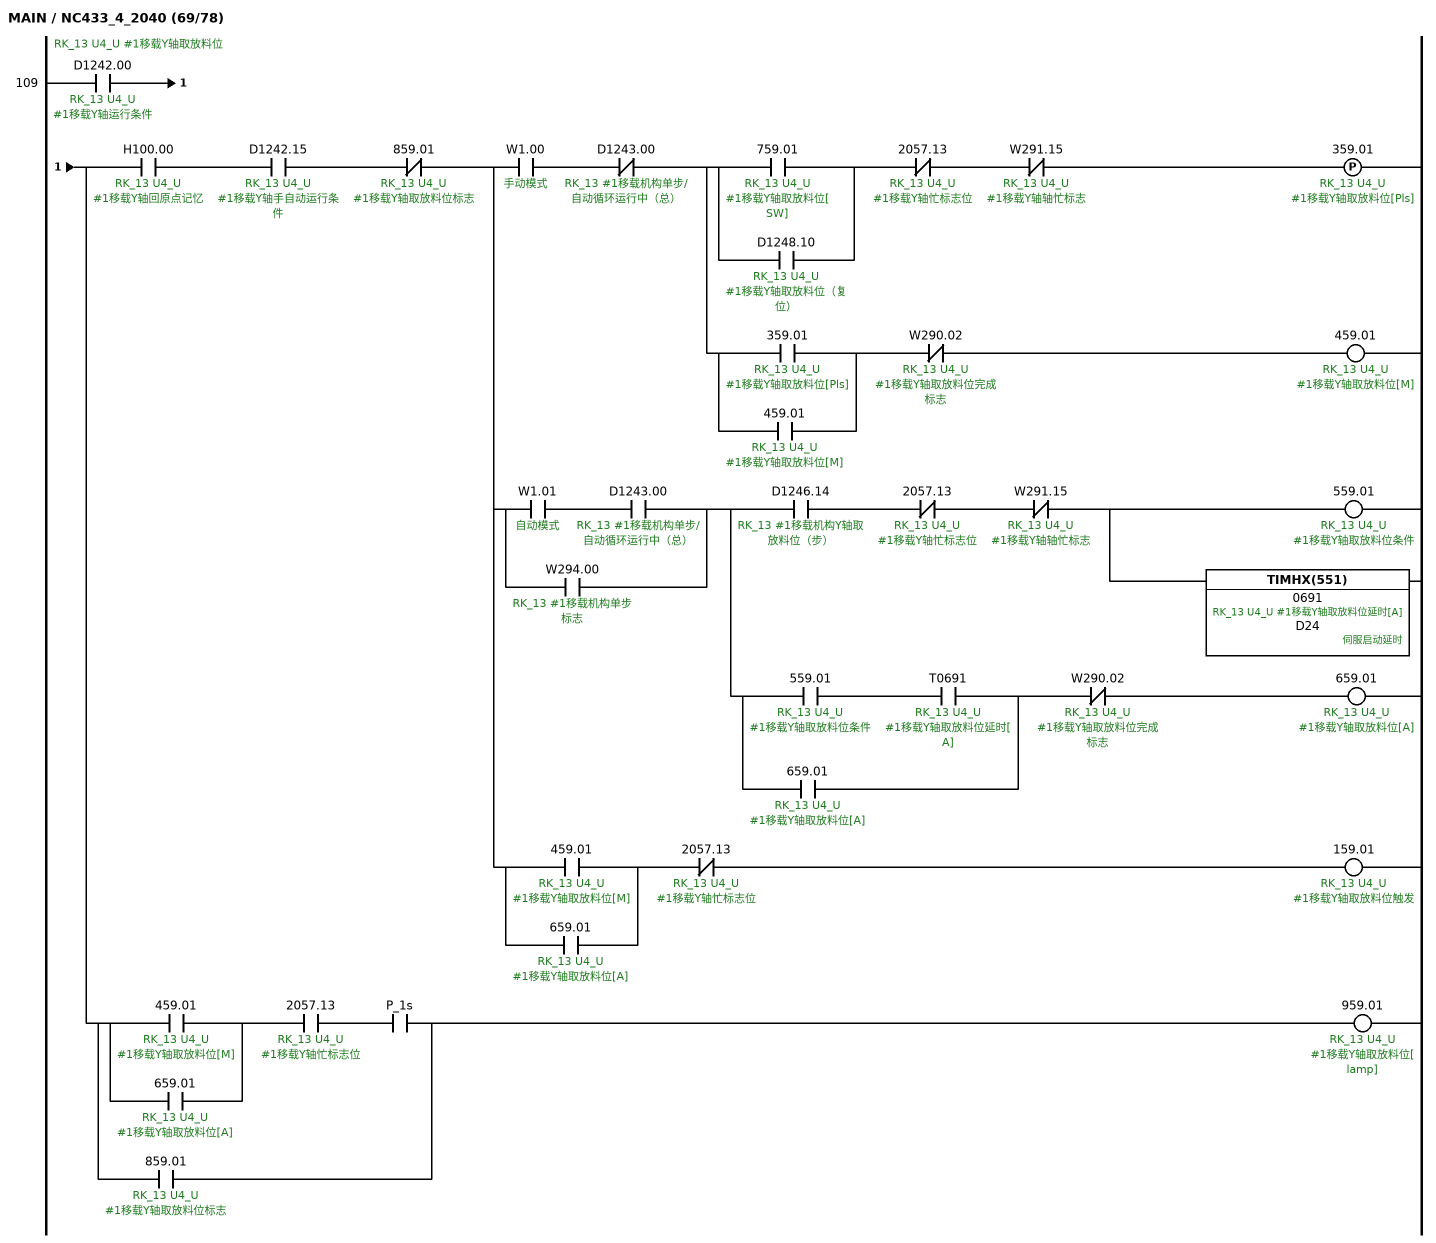
; [picture p216: MAIN / NC433_4_2040, rungs 109-109]
; rung 109: RK_13 U4_U #1移载Y轴取放料位
LD D1242.00  ; RK_13 U4_U #1移载Y轴运行条件
OUT TR0
AND H100.00  ; RK_13 U4_U #1移载Y轴回原点记忆
AND D1242.15  ; RK_13 U4_U #1移载Y轴手自动运行条件
ANDNOT 859.01  ; RK_13 U4_U #1移载Y轴取放料位标志
OUT TR1
AND W1.00  ; 手动模式
ANDNOT D1243.00  ; RK_13 #1移载机构单步/自动循环运行中（总）
OUT TR2
LD 759.01  ; RK_13 U4_U #1移载Y轴取放料位[SW]
OR D1248.10  ; RK_13 U4_U #1移载Y轴取放料位（复位）
ANDLD
ANDNOT 2057.13  ; RK_13 U4_U #1移载Y轴忙标志位
ANDNOT W291.15  ; RK_13 U4_U #1移载Y轴轴忙标志
DIFU(013) 359.01  ; RK_13 U4_U #1移载Y轴取放料位[Pls]
LD TR2
LD 359.01  ; RK_13 U4_U #1移载Y轴取放料位[Pls]
OR 459.01  ; RK_13 U4_U #1移载Y轴取放料位[M]
ANDLD
ANDNOT W290.02  ; RK_13 U4_U #1移载Y轴取放料位完成标志
OUT 459.01  ; RK_13 U4_U #1移载Y轴取放料位[M]
LD TR1
LD W1.01  ; 自动模式
AND D1243.00  ; RK_13 #1移载机构单步/自动循环运行中（总）
OR W294.00  ; RK_13 #1移载机构单步标志
ANDLD
OUT TR2
AND D1246.14  ; RK_13 #1移载机构Y轴取放料位（步）
ANDNOT 2057.13  ; RK_13 U4_U #1移载Y轴忙标志位
ANDNOT W291.15  ; RK_13 U4_U #1移载Y轴轴忙标志
OUT 559.01  ; RK_13 U4_U #1移载Y轴取放料位条件
TIMHX(551) 0691 D24  ; 伺服启动延时, RK_13 U4_U #1移载Y轴取放料位延时[A]
LD TR2
LD 559.01  ; RK_13 U4_U #1移载Y轴取放料位条件
AND T0691  ; RK_13 U4_U #1移载Y轴取放料位延时[A]
OR 659.01  ; RK_13 U4_U #1移载Y轴取放料位[A]
ANDLD
ANDNOT W290.02  ; RK_13 U4_U #1移载Y轴取放料位完成标志
OUT 659.01  ; RK_13 U4_U #1移载Y轴取放料位[A]
LD TR1
LD 459.01  ; RK_13 U4_U #1移载Y轴取放料位[M]
OR 659.01  ; RK_13 U4_U #1移载Y轴取放料位[A]
ANDLD
ANDNOT 2057.13  ; RK_13 U4_U #1移载Y轴忙标志位
OUT 159.01  ; RK_13 U4_U #1移载Y轴取放料位触发
LD TR0
LD 459.01  ; RK_13 U4_U #1移载Y轴取放料位[M]
OR 659.01  ; RK_13 U4_U #1移载Y轴取放料位[A]
AND 2057.13  ; RK_13 U4_U #1移载Y轴忙标志位
AND P_1s
OR 859.01  ; RK_13 U4_U #1移载Y轴取放料位标志
ANDLD
OUT 959.01  ; RK_13 U4_U #1移载Y轴取放料位[lamp]

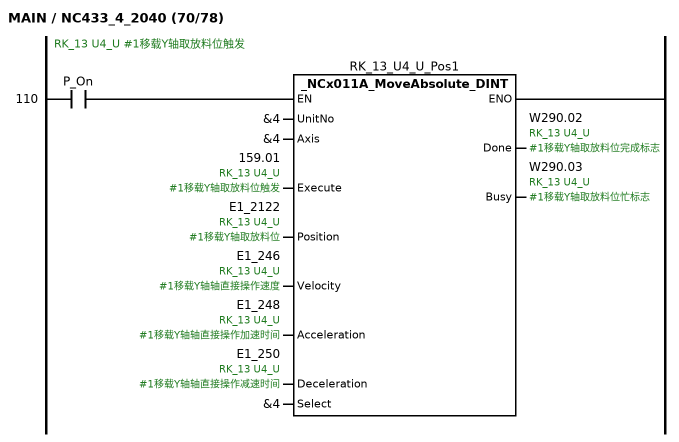
; rung 110: RK_13 U4_U #1移载Y轴取放料位触发
LD P_On
CALL RK_13_U4_U_Pos1 : _NCx011A_MoveAbsolute_DINT (UnitNo := &4, Axis := &4, Execute := 159.01, Position := E1_2122, Velocity := E1_246, Acceleration := E1_248, Deceleration := E1_250, Select := &4, Done => W290.02, Busy => W290.03)  ; RK_13 U4_U #1移载Y轴取放料位触发, RK_13 U4_U #1移载Y轴取放料位, RK_13 U4_U #1移载Y轴轴直接操作速度, RK_13 U4_U #1移载Y轴轴直接操作加速时间, RK_13 U4_U #1移载Y轴轴直接操作减速时间, RK_13 U4_U #1移载Y轴取放料位完成标志, RK_13 U4_U #1移载Y轴取放料位忙标志

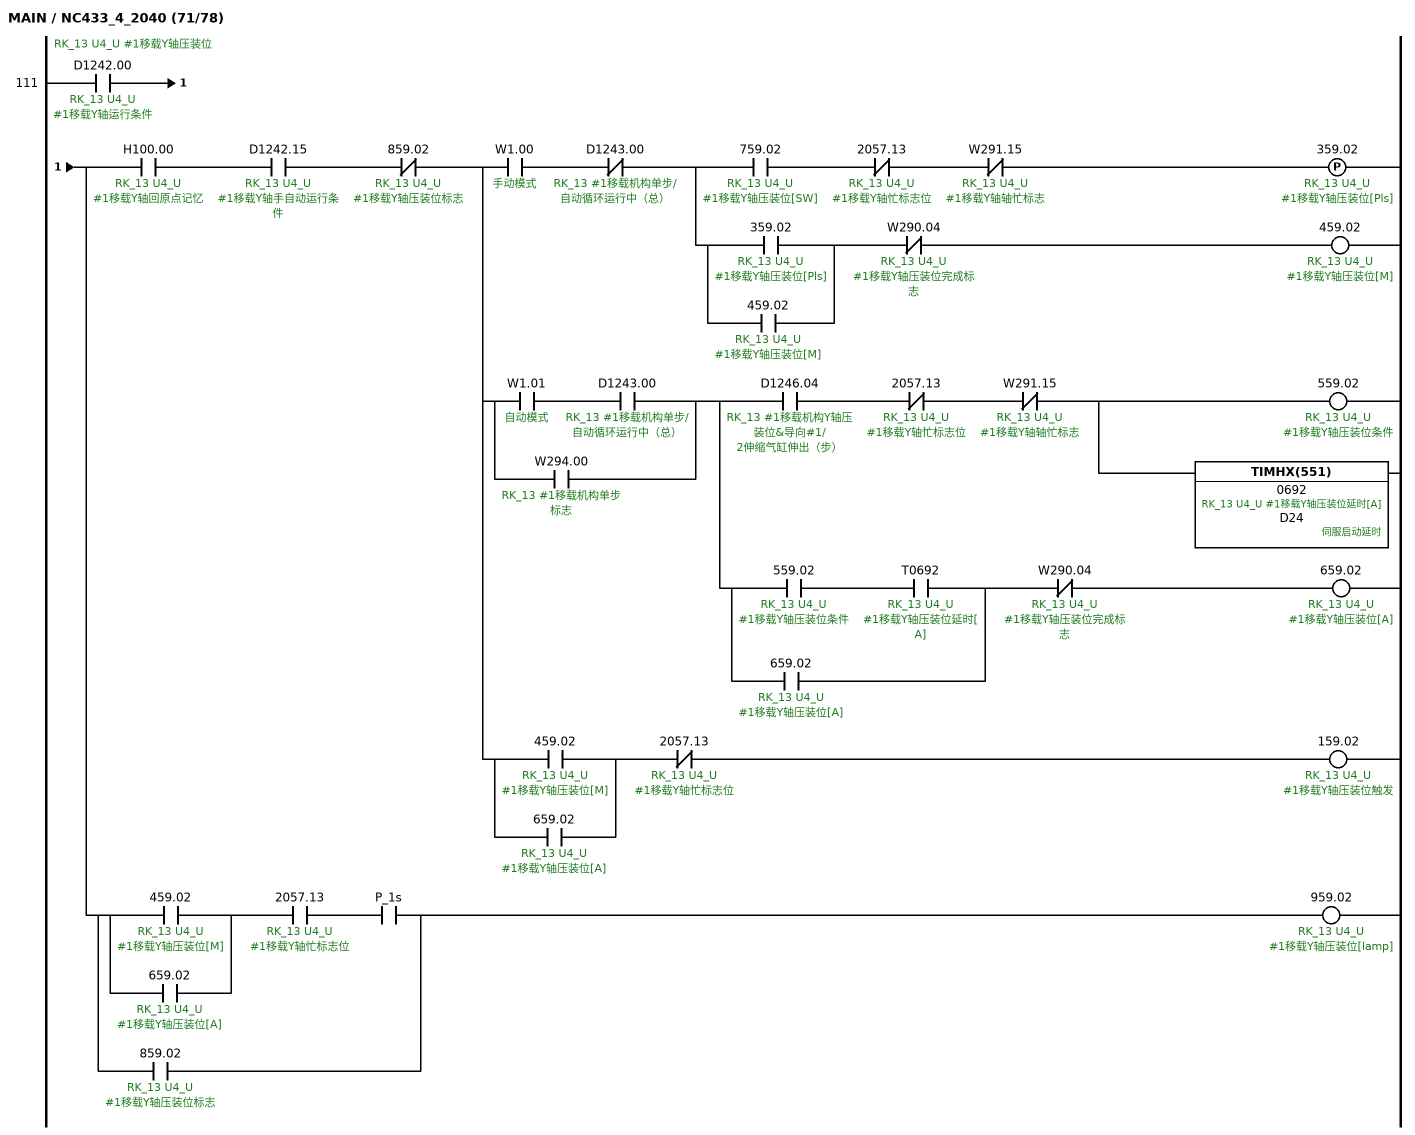
; rung 111: RK_13 U4_U #1移载Y轴压装位
LD D1242.00  ; RK_13 U4_U #1移载Y轴运行条件
OUT TR0
AND H100.00  ; RK_13 U4_U #1移载Y轴回原点记忆
AND D1242.15  ; RK_13 U4_U #1移载Y轴手自动运行条件
ANDNOT 859.02  ; RK_13 U4_U #1移载Y轴压装位标志
OUT TR1
AND W1.00  ; 手动模式
ANDNOT D1243.00  ; RK_13 #1移载机构单步/自动循环运行中（总）
OUT TR2
AND 759.02  ; RK_13 U4_U #1移载Y轴压装位[SW]
ANDNOT 2057.13  ; RK_13 U4_U #1移载Y轴忙标志位
ANDNOT W291.15  ; RK_13 U4_U #1移载Y轴轴忙标志
DIFU(013) 359.02  ; RK_13 U4_U #1移载Y轴压装位[Pls]
LD TR2
LD 359.02  ; RK_13 U4_U #1移载Y轴压装位[Pls]
OR 459.02  ; RK_13 U4_U #1移载Y轴压装位[M]
ANDLD
ANDNOT W290.04  ; RK_13 U4_U #1移载Y轴压装位完成标志
OUT 459.02  ; RK_13 U4_U #1移载Y轴压装位[M]
LD TR1
LD W1.01  ; 自动模式
AND D1243.00  ; RK_13 #1移载机构单步/自动循环运行中（总）
OR W294.00  ; RK_13 #1移载机构单步标志
ANDLD
OUT TR2
AND D1246.04  ; RK_13 #1移载机构Y轴压装位&导向#1/2伸缩气缸伸出（步）
ANDNOT 2057.13  ; RK_13 U4_U #1移载Y轴忙标志位
ANDNOT W291.15  ; RK_13 U4_U #1移载Y轴轴忙标志
OUT 559.02  ; RK_13 U4_U #1移载Y轴压装位条件
TIMHX(551) 0692 D24  ; 伺服启动延时, RK_13 U4_U #1移载Y轴压装位延时[A]
LD TR2
LD 559.02  ; RK_13 U4_U #1移载Y轴压装位条件
AND T0692  ; RK_13 U4_U #1移载Y轴压装位延时[A]
OR 659.02  ; RK_13 U4_U #1移载Y轴压装位[A]
ANDLD
ANDNOT W290.04  ; RK_13 U4_U #1移载Y轴压装位完成标志
OUT 659.02  ; RK_13 U4_U #1移载Y轴压装位[A]
LD TR1
LD 459.02  ; RK_13 U4_U #1移载Y轴压装位[M]
OR 659.02  ; RK_13 U4_U #1移载Y轴压装位[A]
ANDLD
ANDNOT 2057.13  ; RK_13 U4_U #1移载Y轴忙标志位
OUT 159.02  ; RK_13 U4_U #1移载Y轴压装位触发
LD TR0
LD 459.02  ; RK_13 U4_U #1移载Y轴压装位[M]
OR 659.02  ; RK_13 U4_U #1移载Y轴压装位[A]
AND 2057.13  ; RK_13 U4_U #1移载Y轴忙标志位
AND P_1s
OR 859.02  ; RK_13 U4_U #1移载Y轴压装位标志
ANDLD
OUT 959.02  ; RK_13 U4_U #1移载Y轴压装位[lamp]

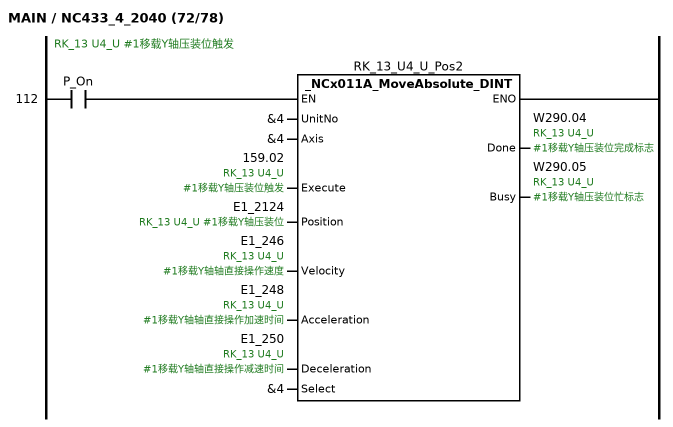
; rung 112: RK_13 U4_U #1移载Y轴压装位触发
LD P_On
CALL RK_13_U4_U_Pos2 : _NCx011A_MoveAbsolute_DINT (UnitNo := &4, Axis := &4, Execute := 159.02, Position := E1_2124, Velocity := E1_246, Acceleration := E1_248, Deceleration := E1_250, Select := &4, Done => W290.04, Busy => W290.05)  ; RK_13 U4_U #1移载Y轴压装位触发, RK_13 U4_U #1移载Y轴压装位, RK_13 U4_U #1移载Y轴轴直接操作速度, RK_13 U4_U #1移载Y轴轴直接操作加速时间, RK_13 U4_U #1移载Y轴轴直接操作减速时间, RK_13 U4_U #1移载Y轴压装位完成标志, RK_13 U4_U #1移载Y轴压装位忙标志

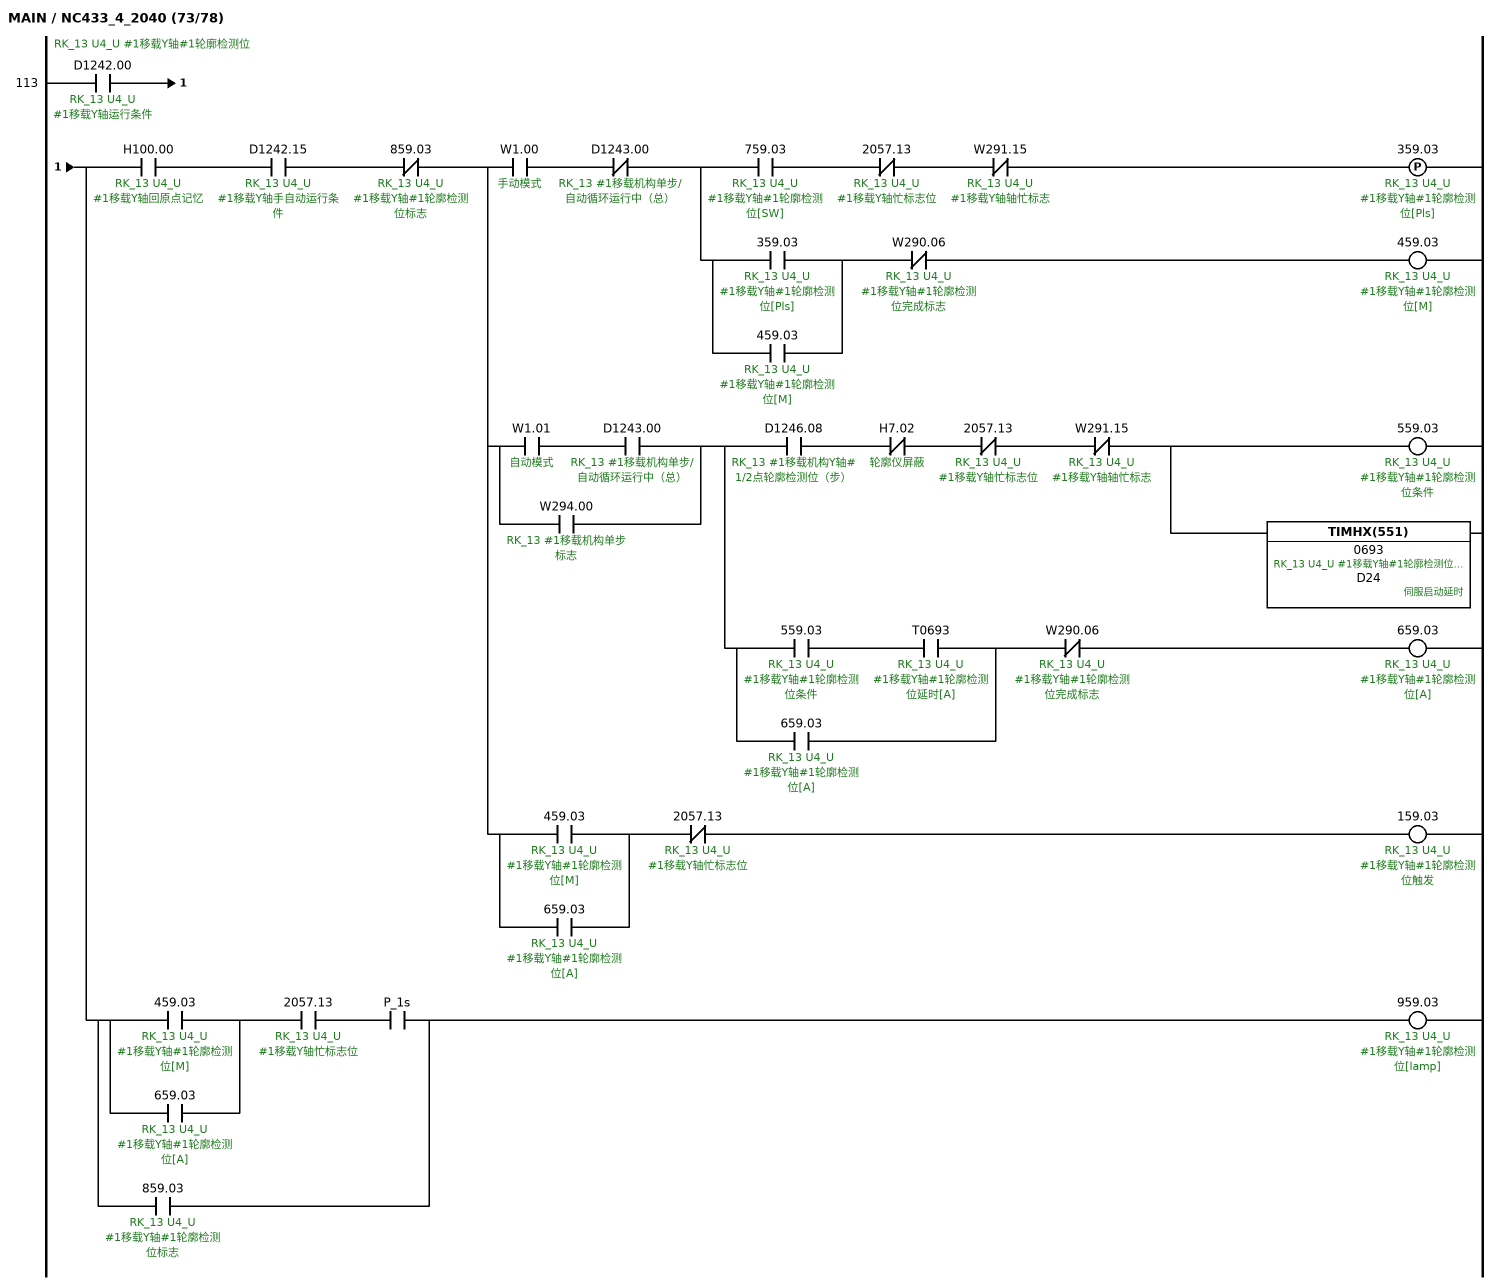
; rung 113: RK_13 U4_U #1移载Y轴#1轮廓检测位
LD D1242.00  ; RK_13 U4_U #1移载Y轴运行条件
OUT TR0
AND H100.00  ; RK_13 U4_U #1移载Y轴回原点记忆
AND D1242.15  ; RK_13 U4_U #1移载Y轴手自动运行条件
ANDNOT 859.03  ; RK_13 U4_U #1移载Y轴#1轮廓检测位标志
OUT TR1
AND W1.00  ; 手动模式
ANDNOT D1243.00  ; RK_13 #1移载机构单步/自动循环运行中（总）
OUT TR2
AND 759.03  ; RK_13 U4_U #1移载Y轴#1轮廓检测位[SW]
ANDNOT 2057.13  ; RK_13 U4_U #1移载Y轴忙标志位
ANDNOT W291.15  ; RK_13 U4_U #1移载Y轴轴忙标志
DIFU(013) 359.03  ; RK_13 U4_U #1移载Y轴#1轮廓检测位[Pls]
LD TR2
LD 359.03  ; RK_13 U4_U #1移载Y轴#1轮廓检测位[Pls]
OR 459.03  ; RK_13 U4_U #1移载Y轴#1轮廓检测位[M]
ANDLD
ANDNOT W290.06  ; RK_13 U4_U #1移载Y轴#1轮廓检测位完成标志
OUT 459.03  ; RK_13 U4_U #1移载Y轴#1轮廓检测位[M]
LD TR1
LD W1.01  ; 自动模式
AND D1243.00  ; RK_13 #1移载机构单步/自动循环运行中（总）
OR W294.00  ; RK_13 #1移载机构单步标志
ANDLD
OUT TR2
AND D1246.08  ; RK_13 #1移载机构Y轴#1/2点轮廓检测位（步）
ANDNOT H7.02  ; 轮廓仪屏蔽
ANDNOT 2057.13  ; RK_13 U4_U #1移载Y轴忙标志位
ANDNOT W291.15  ; RK_13 U4_U #1移载Y轴轴忙标志
OUT 559.03  ; RK_13 U4_U #1移载Y轴#1轮廓检测位条件
TIMHX(551) 0693 D24  ; 伺服启动延时, RK_13 U4_U #1移载Y轴#1轮廓检测位延时[A]
LD TR2
LD 559.03  ; RK_13 U4_U #1移载Y轴#1轮廓检测位条件
AND T0693  ; RK_13 U4_U #1移载Y轴#1轮廓检测位延时[A]
OR 659.03  ; RK_13 U4_U #1移载Y轴#1轮廓检测位[A]
ANDLD
ANDNOT W290.06  ; RK_13 U4_U #1移载Y轴#1轮廓检测位完成标志
OUT 659.03  ; RK_13 U4_U #1移载Y轴#1轮廓检测位[A]
LD TR1
LD 459.03  ; RK_13 U4_U #1移载Y轴#1轮廓检测位[M]
OR 659.03  ; RK_13 U4_U #1移载Y轴#1轮廓检测位[A]
ANDLD
ANDNOT 2057.13  ; RK_13 U4_U #1移载Y轴忙标志位
OUT 159.03  ; RK_13 U4_U #1移载Y轴#1轮廓检测位触发
LD TR0
LD 459.03  ; RK_13 U4_U #1移载Y轴#1轮廓检测位[M]
OR 659.03  ; RK_13 U4_U #1移载Y轴#1轮廓检测位[A]
AND 2057.13  ; RK_13 U4_U #1移载Y轴忙标志位
AND P_1s
OR 859.03  ; RK_13 U4_U #1移载Y轴#1轮廓检测位标志
ANDLD
OUT 959.03  ; RK_13 U4_U #1移载Y轴#1轮廓检测位[lamp]

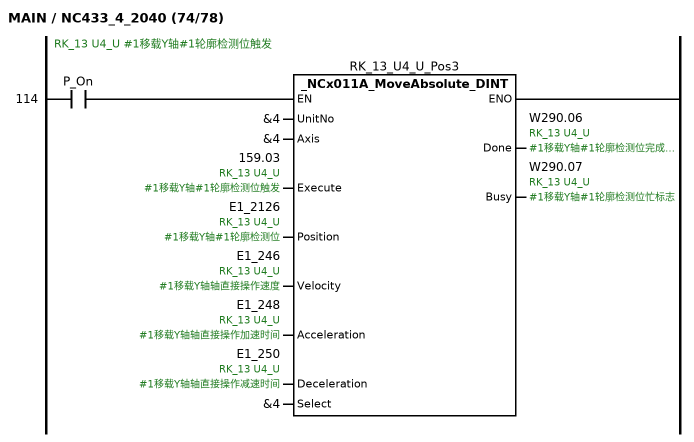
; rung 114: RK_13 U4_U #1移载Y轴#1轮廓检测位触发
LD P_On
CALL RK_13_U4_U_Pos3 : _NCx011A_MoveAbsolute_DINT (UnitNo := &4, Axis := &4, Execute := 159.03, Position := E1_2126, Velocity := E1_246, Acceleration := E1_248, Deceleration := E1_250, Select := &4, Done => W290.06, Busy => W290.07)  ; RK_13 U4_U #1移载Y轴#1轮廓检测位触发, RK_13 U4_U #1移载Y轴#1轮廓检测位, RK_13 U4_U #1移载Y轴轴直接操作速度, RK_13 U4_U #1移载Y轴轴直接操作加速时间, RK_13 U4_U #1移载Y轴轴直接操作减速时间, RK_13 U4_U #1移载Y轴#1轮廓检测位完成标志, RK_13 U4_U #1移载Y轴#1轮廓检测位忙标志

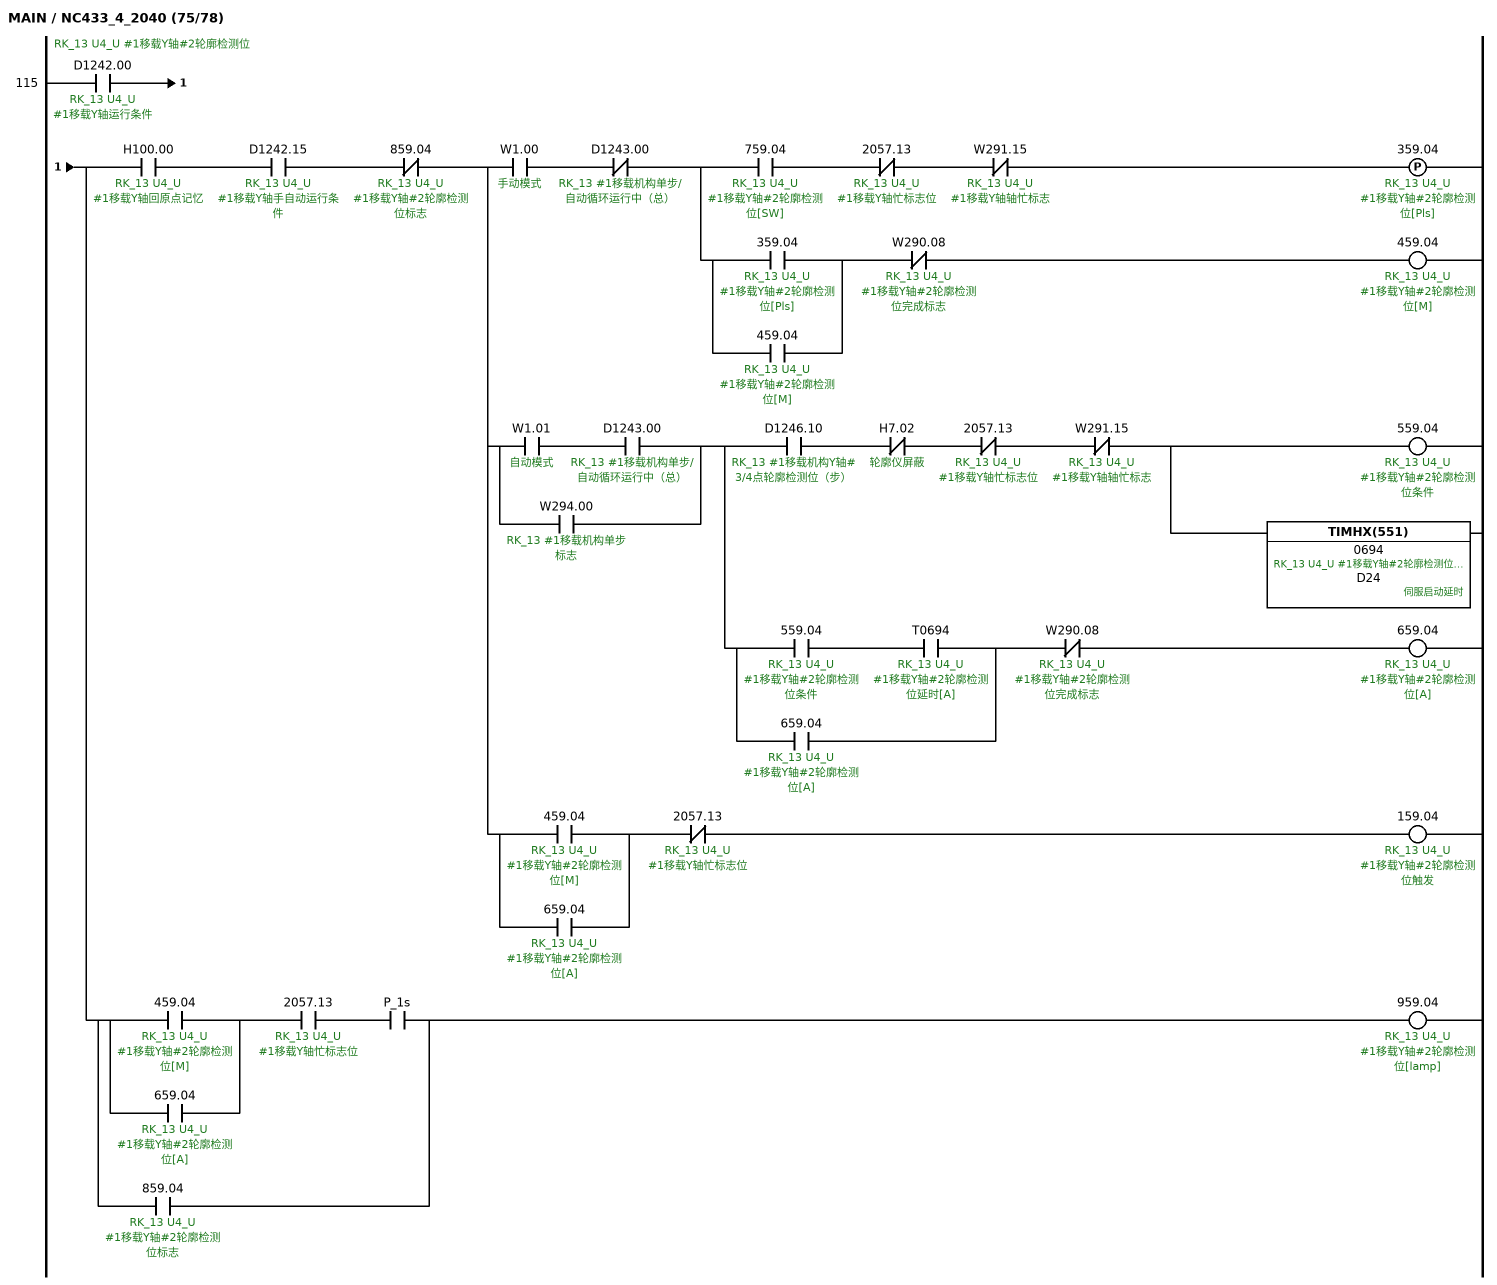
; rung 115: RK_13 U4_U #1移载Y轴#2轮廓检测位
LD D1242.00  ; RK_13 U4_U #1移载Y轴运行条件
OUT TR0
AND H100.00  ; RK_13 U4_U #1移载Y轴回原点记忆
AND D1242.15  ; RK_13 U4_U #1移载Y轴手自动运行条件
ANDNOT 859.04  ; RK_13 U4_U #1移载Y轴#2轮廓检测位标志
OUT TR1
AND W1.00  ; 手动模式
ANDNOT D1243.00  ; RK_13 #1移载机构单步/自动循环运行中（总）
OUT TR2
AND 759.04  ; RK_13 U4_U #1移载Y轴#2轮廓检测位[SW]
ANDNOT 2057.13  ; RK_13 U4_U #1移载Y轴忙标志位
ANDNOT W291.15  ; RK_13 U4_U #1移载Y轴轴忙标志
DIFU(013) 359.04  ; RK_13 U4_U #1移载Y轴#2轮廓检测位[Pls]
LD TR2
LD 359.04  ; RK_13 U4_U #1移载Y轴#2轮廓检测位[Pls]
OR 459.04  ; RK_13 U4_U #1移载Y轴#2轮廓检测位[M]
ANDLD
ANDNOT W290.08  ; RK_13 U4_U #1移载Y轴#2轮廓检测位完成标志
OUT 459.04  ; RK_13 U4_U #1移载Y轴#2轮廓检测位[M]
LD TR1
LD W1.01  ; 自动模式
AND D1243.00  ; RK_13 #1移载机构单步/自动循环运行中（总）
OR W294.00  ; RK_13 #1移载机构单步标志
ANDLD
OUT TR2
AND D1246.10  ; RK_13 #1移载机构Y轴#3/4点轮廓检测位（步）
ANDNOT H7.02  ; 轮廓仪屏蔽
ANDNOT 2057.13  ; RK_13 U4_U #1移载Y轴忙标志位
ANDNOT W291.15  ; RK_13 U4_U #1移载Y轴轴忙标志
OUT 559.04  ; RK_13 U4_U #1移载Y轴#2轮廓检测位条件
TIMHX(551) 0694 D24  ; 伺服启动延时, RK_13 U4_U #1移载Y轴#2轮廓检测位延时[A]
LD TR2
LD 559.04  ; RK_13 U4_U #1移载Y轴#2轮廓检测位条件
AND T0694  ; RK_13 U4_U #1移载Y轴#2轮廓检测位延时[A]
OR 659.04  ; RK_13 U4_U #1移载Y轴#2轮廓检测位[A]
ANDLD
ANDNOT W290.08  ; RK_13 U4_U #1移载Y轴#2轮廓检测位完成标志
OUT 659.04  ; RK_13 U4_U #1移载Y轴#2轮廓检测位[A]
LD TR1
LD 459.04  ; RK_13 U4_U #1移载Y轴#2轮廓检测位[M]
OR 659.04  ; RK_13 U4_U #1移载Y轴#2轮廓检测位[A]
ANDLD
ANDNOT 2057.13  ; RK_13 U4_U #1移载Y轴忙标志位
OUT 159.04  ; RK_13 U4_U #1移载Y轴#2轮廓检测位触发
LD TR0
LD 459.04  ; RK_13 U4_U #1移载Y轴#2轮廓检测位[M]
OR 659.04  ; RK_13 U4_U #1移载Y轴#2轮廓检测位[A]
AND 2057.13  ; RK_13 U4_U #1移载Y轴忙标志位
AND P_1s
OR 859.04  ; RK_13 U4_U #1移载Y轴#2轮廓检测位标志
ANDLD
OUT 959.04  ; RK_13 U4_U #1移载Y轴#2轮廓检测位[lamp]

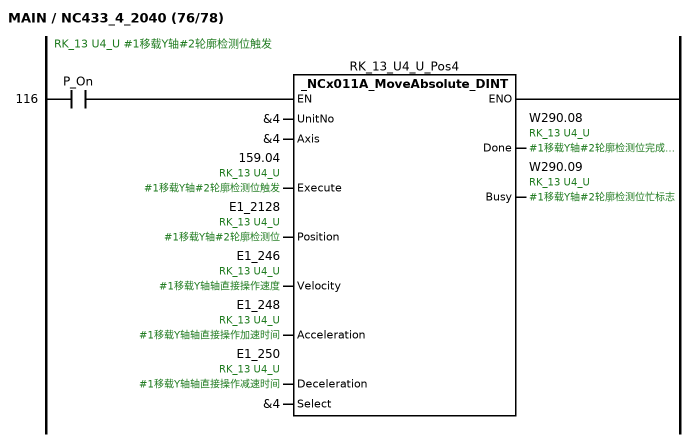
; rung 116: RK_13 U4_U #1移载Y轴#2轮廓检测位触发
LD P_On
CALL RK_13_U4_U_Pos4 : _NCx011A_MoveAbsolute_DINT (UnitNo := &4, Axis := &4, Execute := 159.04, Position := E1_2128, Velocity := E1_246, Acceleration := E1_248, Deceleration := E1_250, Select := &4, Done => W290.08, Busy => W290.09)  ; RK_13 U4_U #1移载Y轴#2轮廓检测位触发, RK_13 U4_U #1移载Y轴#2轮廓检测位, RK_13 U4_U #1移载Y轴轴直接操作速度, RK_13 U4_U #1移载Y轴轴直接操作加速时间, RK_13 U4_U #1移载Y轴轴直接操作减速时间, RK_13 U4_U #1移载Y轴#2轮廓检测位完成标志, RK_13 U4_U #1移载Y轴#2轮廓检测位忙标志

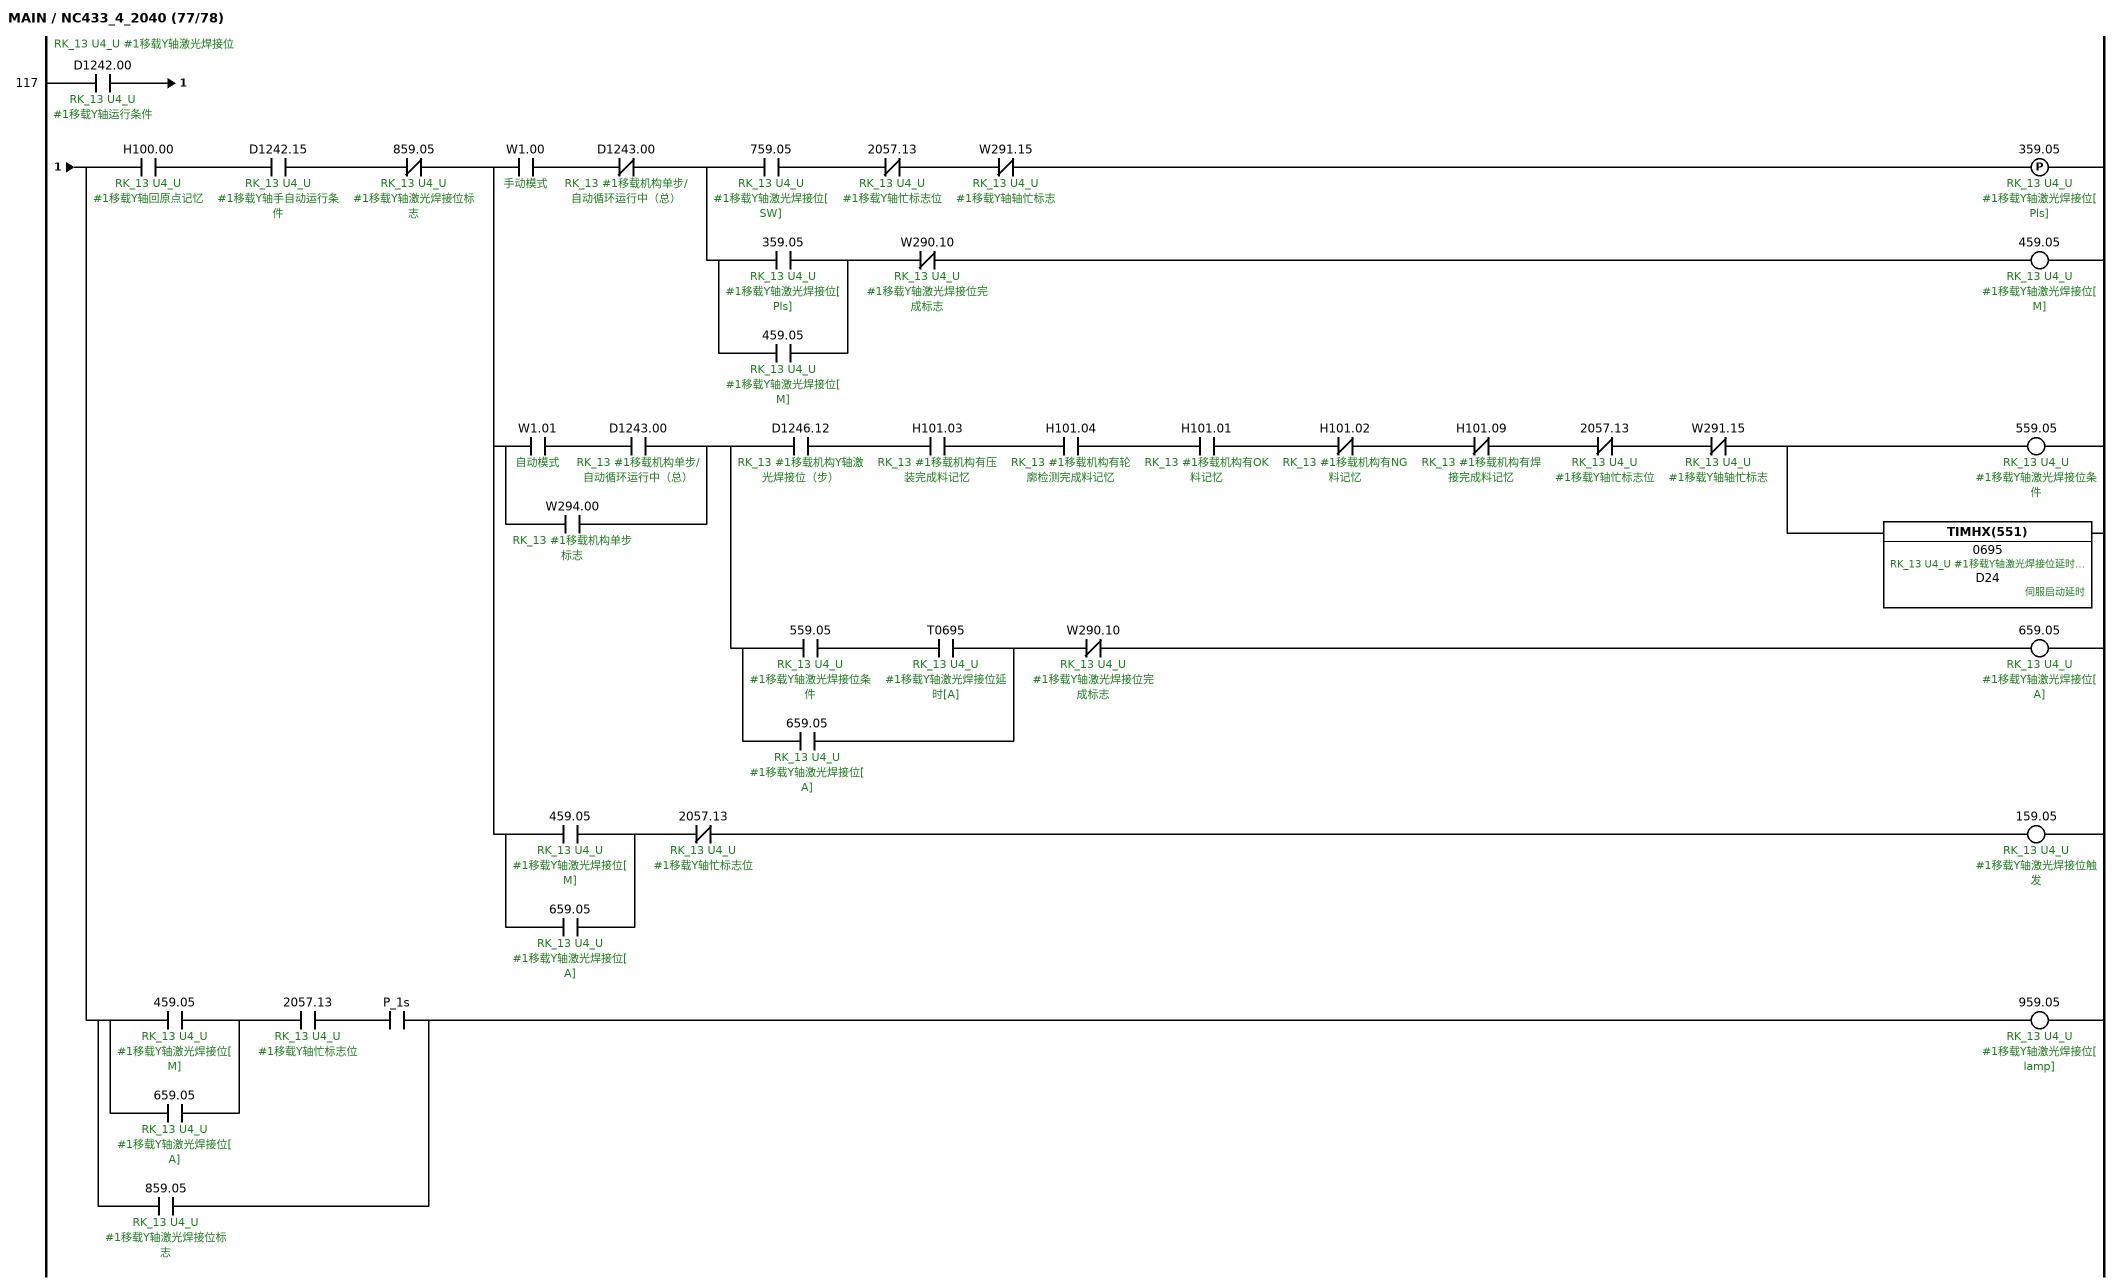
; rung 117: RK_13 U4_U #1移载Y轴激光焊接位
LD D1242.00  ; RK_13 U4_U #1移载Y轴运行条件
OUT TR0
AND H100.00  ; RK_13 U4_U #1移载Y轴回原点记忆
AND D1242.15  ; RK_13 U4_U #1移载Y轴手自动运行条件
ANDNOT 859.05  ; RK_13 U4_U #1移载Y轴激光焊接位标志
OUT TR1
AND W1.00  ; 手动模式
ANDNOT D1243.00  ; RK_13 #1移载机构单步/自动循环运行中（总）
OUT TR2
AND 759.05  ; RK_13 U4_U #1移载Y轴激光焊接位[SW]
ANDNOT 2057.13  ; RK_13 U4_U #1移载Y轴忙标志位
ANDNOT W291.15  ; RK_13 U4_U #1移载Y轴轴忙标志
DIFU(013) 359.05  ; RK_13 U4_U #1移载Y轴激光焊接位[Pls]
LD TR2
LD 359.05  ; RK_13 U4_U #1移载Y轴激光焊接位[Pls]
OR 459.05  ; RK_13 U4_U #1移载Y轴激光焊接位[M]
ANDLD
ANDNOT W290.10  ; RK_13 U4_U #1移载Y轴激光焊接位完成标志
OUT 459.05  ; RK_13 U4_U #1移载Y轴激光焊接位[M]
LD TR1
LD W1.01  ; 自动模式
AND D1243.00  ; RK_13 #1移载机构单步/自动循环运行中（总）
OR W294.00  ; RK_13 #1移载机构单步标志
ANDLD
OUT TR2
AND D1246.12  ; RK_13 #1移载机构Y轴激光焊接位（步）
AND H101.03  ; RK_13 #1移载机构有压装完成料记忆
AND H101.04  ; RK_13 #1移载机构有轮廓检测完成料记忆
AND H101.01  ; RK_13 #1移载机构有OK料记忆
ANDNOT H101.02  ; RK_13 #1移载机构有NG料记忆
ANDNOT H101.09  ; RK_13 #1移载机构有焊接完成料记忆
ANDNOT 2057.13  ; RK_13 U4_U #1移载Y轴忙标志位
ANDNOT W291.15  ; RK_13 U4_U #1移载Y轴轴忙标志
OUT 559.05  ; RK_13 U4_U #1移载Y轴激光焊接位条件
TIMHX(551) 0695 D24  ; 伺服启动延时, RK_13 U4_U #1移载Y轴激光焊接位延时[A]
LD TR2
LD 559.05  ; RK_13 U4_U #1移载Y轴激光焊接位条件
AND T0695  ; RK_13 U4_U #1移载Y轴激光焊接位延时[A]
OR 659.05  ; RK_13 U4_U #1移载Y轴激光焊接位[A]
ANDLD
ANDNOT W290.10  ; RK_13 U4_U #1移载Y轴激光焊接位完成标志
OUT 659.05  ; RK_13 U4_U #1移载Y轴激光焊接位[A]
LD TR1
LD 459.05  ; RK_13 U4_U #1移载Y轴激光焊接位[M]
OR 659.05  ; RK_13 U4_U #1移载Y轴激光焊接位[A]
ANDLD
ANDNOT 2057.13  ; RK_13 U4_U #1移载Y轴忙标志位
OUT 159.05  ; RK_13 U4_U #1移载Y轴激光焊接位触发
LD TR0
LD 459.05  ; RK_13 U4_U #1移载Y轴激光焊接位[M]
OR 659.05  ; RK_13 U4_U #1移载Y轴激光焊接位[A]
AND 2057.13  ; RK_13 U4_U #1移载Y轴忙标志位
AND P_1s
OR 859.05  ; RK_13 U4_U #1移载Y轴激光焊接位标志
ANDLD
OUT 959.05  ; RK_13 U4_U #1移载Y轴激光焊接位[lamp]

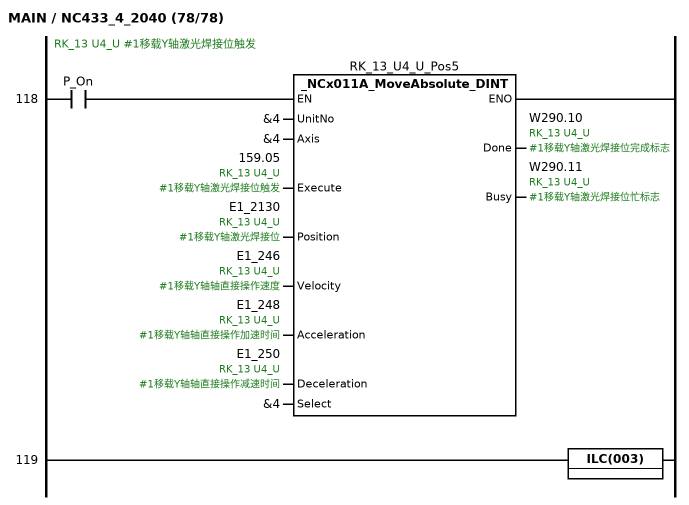
; rung 118: RK_13 U4_U #1移载Y轴激光焊接位触发
LD P_On
CALL RK_13_U4_U_Pos5 : _NCx011A_MoveAbsolute_DINT (UnitNo := &4, Axis := &4, Execute := 159.05, Position := E1_2130, Velocity := E1_246, Acceleration := E1_248, Deceleration := E1_250, Select := &4, Done => W290.10, Busy => W290.11)  ; RK_13 U4_U #1移载Y轴激光焊接位触发, RK_13 U4_U #1移载Y轴激光焊接位, RK_13 U4_U #1移载Y轴轴直接操作速度, RK_13 U4_U #1移载Y轴轴直接操作加速时间, RK_13 U4_U #1移载Y轴轴直接操作减速时间, RK_13 U4_U #1移载Y轴激光焊接位完成标志, RK_13 U4_U #1移载Y轴激光焊接位忙标志
; rung 119
ILC(003)

### Section NC433_6_2060

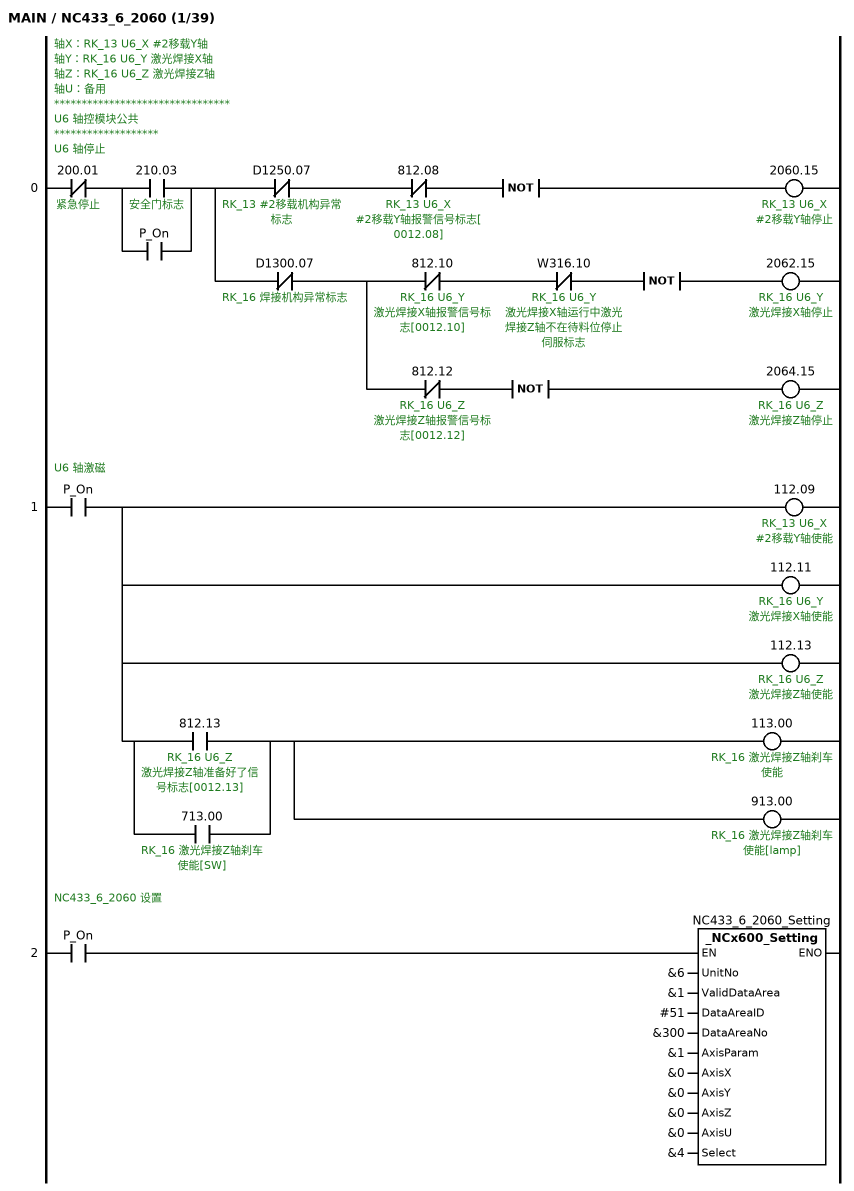
; rung 0: 轴X：RK_13 U6_X #2移载Y轴 / 轴Y：RK_16 U6_Y 激光焊接X轴 / 轴Z：RK_16 U6_Z 激光焊接Z轴 / 轴U：备用 / ******************************** / U6 轴控模块公共 / ******************* / U6 轴停止
LDNOT 200.01  ; 紧急停止
LD 210.03  ; 安全门标志
OR P_On
ANDLD
OUT TR0
ANDNOT D1250.07  ; RK_13 #2移载机构异常标志
ANDNOT 812.08  ; RK_13 U6_X #2移载Y轴报警信号标志[0012.08]
NOT(520)
OUT 2060.15  ; RK_13 U6_X #2移载Y轴停止
LD TR0
ANDNOT D1300.07  ; RK_16 焊接机构异常标志
OUT TR0
ANDNOT 812.10  ; RK_16 U6_Y 激光焊接X轴报警信号标志[0012.10]
ANDNOT W316.10  ; RK_16 U6_Y 激光焊接X轴运行中激光焊接Z轴不在待料位停止伺服标志
NOT(520)
OUT 2062.15  ; RK_16 U6_Y 激光焊接X轴停止
LD TR0
ANDNOT 812.12  ; RK_16 U6_Z 激光焊接Z轴报警信号标志[0012.12]
NOT(520)
OUT 2064.15  ; RK_16 U6_Z 激光焊接Z轴停止
; rung 1: U6 轴激磁
LD P_On
OUT 112.09  ; RK_13 U6_X #2移载Y轴使能
OUT 112.11  ; RK_16 U6_Y 激光焊接X轴使能
OUT 112.13  ; RK_16 U6_Z 激光焊接Z轴使能
LD 812.13  ; RK_16 U6_Z 激光焊接Z轴准备好了信号标志[0012.13]
OR 713.00  ; RK_16 激光焊接Z轴刹车使能[SW]
ANDLD
OUT 113.00  ; RK_16 激光焊接Z轴刹车使能
OUT 913.00  ; RK_16 激光焊接Z轴刹车使能[lamp]
; rung 2: NC433_6_2060 设置
LD P_On
CALL NC433_6_2060_Setting : _NCx600_Setting (UnitNo := &6, ValidDataArea := &1, DataAreaID := #51, DataAreaNo := &300, AxisParam := &1, AxisX := &0, AxisY := &0, AxisZ := &0, AxisU := &0, Select := &4)

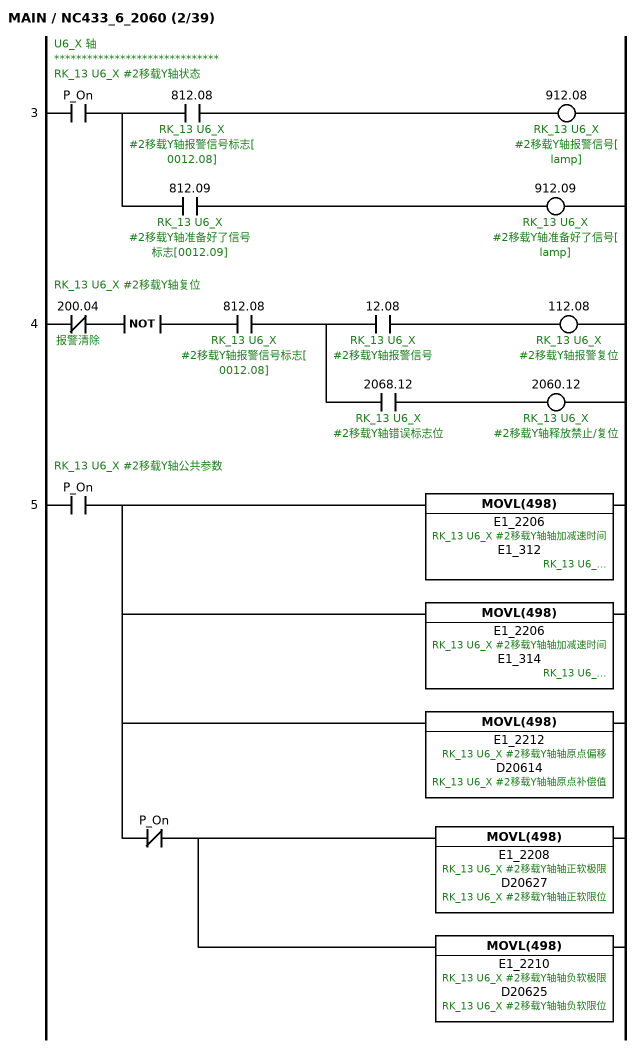
; rung 3: U6_X 轴 / ****************************** / RK_13 U6_X #2移载Y轴状态
LD P_On
OUT TR0
AND 812.08  ; RK_13 U6_X #2移载Y轴报警信号标志[0012.08]
OUT 912.08  ; RK_13 U6_X #2移载Y轴报警信号[lamp]
LD TR0
AND 812.09  ; RK_13 U6_X #2移载Y轴准备好了信号标志[0012.09]
OUT 912.09  ; RK_13 U6_X #2移载Y轴准备好了信号[lamp]
; rung 4: RK_13 U6_X #2移载Y轴复位
LDNOT 200.04  ; 报警清除
NOT(520)
AND 812.08  ; RK_13 U6_X #2移载Y轴报警信号标志[0012.08]
OUT TR0
AND 12.08  ; RK_13 U6_X #2移载Y轴报警信号
OUT 112.08  ; RK_13 U6_X #2移载Y轴报警复位
LD TR0
AND 2068.12  ; RK_13 U6_X #2移载Y轴错误标志位
OUT 2060.12  ; RK_13 U6_X #2移载Y轴释放禁止/复位
; rung 5: RK_13 U6_X #2移载Y轴公共参数
LD P_On
MOVL(498) E1_2206 E1_312  ; RK_13 U6_X #2移载Y轴轴加减速时间, RK_13 U6_X #2移载Y轴X轴直接操作加速时间
MOVL(498) E1_2206 E1_314  ; RK_13 U6_X #2移载Y轴轴加减速时间, RK_13 U6_X #2移载Y轴轴直接操作减速时间
MOVL(498) E1_2212 D20614  ; RK_13 U6_X #2移载Y轴轴原点偏移, RK_13 U6_X #2移载Y轴轴原点补偿值
ANDNOT P_On
MOVL(498) E1_2208 D20627  ; RK_13 U6_X #2移载Y轴轴正软极限, RK_13 U6_X #2移载Y轴轴正软限位
MOVL(498) E1_2210 D20625  ; RK_13 U6_X #2移载Y轴轴负软极限, RK_13 U6_X #2移载Y轴轴负软限位

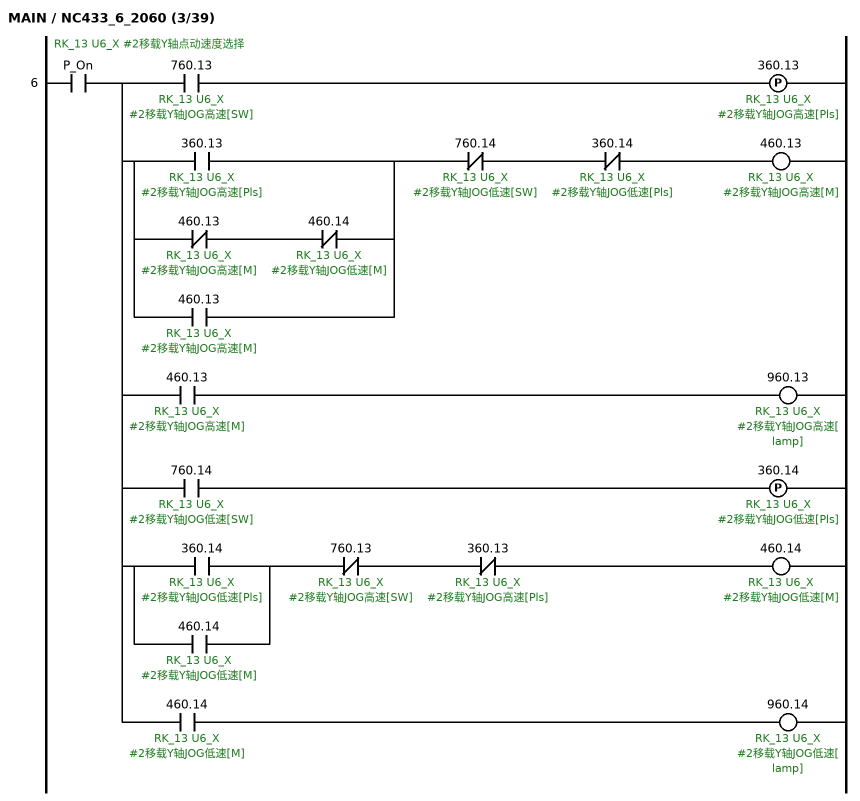
; rung 6: RK_13 U6_X #2移载Y轴点动速度选择
LD P_On
OUT TR0
AND 760.13  ; RK_13 U6_X #2移载Y轴JOG高速[SW]
DIFU(013) 360.13  ; RK_13 U6_X #2移载Y轴JOG高速[Pls]
LD TR0
LD 360.13  ; RK_13 U6_X #2移载Y轴JOG高速[Pls]
LDNOT 460.13  ; RK_13 U6_X #2移载Y轴JOG高速[M]
ANDNOT 460.14  ; RK_13 U6_X #2移载Y轴JOG低速[M]
ORLD
OR 460.13  ; RK_13 U6_X #2移载Y轴JOG高速[M]
ANDLD
ANDNOT 760.14  ; RK_13 U6_X #2移载Y轴JOG低速[SW]
ANDNOT 360.14  ; RK_13 U6_X #2移载Y轴JOG低速[Pls]
OUT 460.13  ; RK_13 U6_X #2移载Y轴JOG高速[M]
LD TR0
AND 460.13  ; RK_13 U6_X #2移载Y轴JOG高速[M]
OUT 960.13  ; RK_13 U6_X #2移载Y轴JOG高速[lamp]
LD TR0
AND 760.14  ; RK_13 U6_X #2移载Y轴JOG低速[SW]
DIFU(013) 360.14  ; RK_13 U6_X #2移载Y轴JOG低速[Pls]
LD TR0
LD 360.14  ; RK_13 U6_X #2移载Y轴JOG低速[Pls]
OR 460.14  ; RK_13 U6_X #2移载Y轴JOG低速[M]
ANDLD
ANDNOT 760.13  ; RK_13 U6_X #2移载Y轴JOG高速[SW]
ANDNOT 360.13  ; RK_13 U6_X #2移载Y轴JOG高速[Pls]
OUT 460.14  ; RK_13 U6_X #2移载Y轴JOG低速[M]
LD TR0
AND 460.14  ; RK_13 U6_X #2移载Y轴JOG低速[M]
OUT 960.14  ; RK_13 U6_X #2移载Y轴JOG低速[lamp]

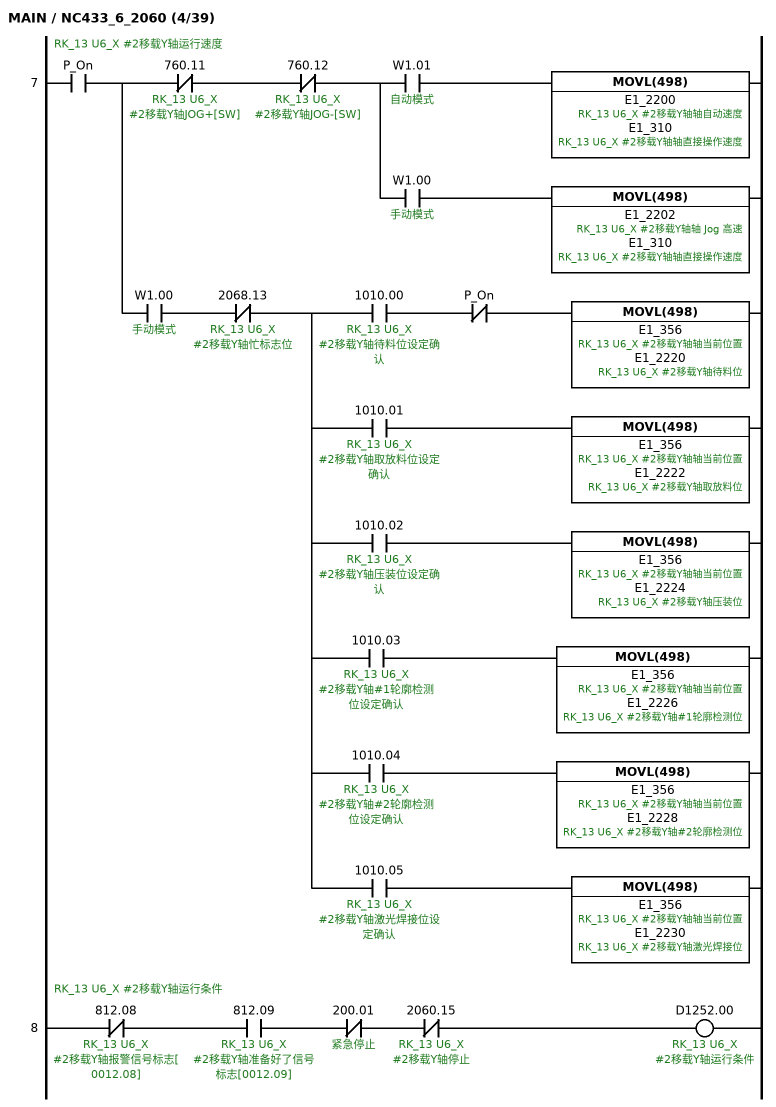
; rung 7: RK_13 U6_X #2移载Y轴运行速度
LD P_On
OUT TR0
ANDNOT 760.11  ; RK_13 U6_X #2移载Y轴JOG+[SW]
ANDNOT 760.12  ; RK_13 U6_X #2移载Y轴JOG-[SW]
OUT TR1
AND W1.01  ; 自动模式
MOVL(498) E1_2200 E1_310  ; RK_13 U6_X #2移载Y轴轴自动速度, RK_13 U6_X #2移载Y轴轴直接操作速度
LD TR1
AND W1.00  ; 手动模式
MOVL(498) E1_2202 E1_310  ; RK_13 U6_X #2移载Y轴轴 Jog 高速, RK_13 U6_X #2移载Y轴轴直接操作速度
LD TR0
AND W1.00  ; 手动模式
ANDNOT 2068.13  ; RK_13 U6_X #2移载Y轴忙标志位
OUT TR0
AND 1010.00  ; RK_13 U6_X #2移载Y轴待料位设定确认
ANDNOT P_On
MOVL(498) E1_356 E1_2220  ; RK_13 U6_X #2移载Y轴轴当前位置, RK_13 U6_X #2移载Y轴待料位
LD TR0
AND 1010.01  ; RK_13 U6_X #2移载Y轴取放料位设定确认
MOVL(498) E1_356 E1_2222  ; RK_13 U6_X #2移载Y轴轴当前位置, RK_13 U6_X #2移载Y轴取放料位
LD TR0
AND 1010.02  ; RK_13 U6_X #2移载Y轴压装位设定确认
MOVL(498) E1_356 E1_2224  ; RK_13 U6_X #2移载Y轴轴当前位置, RK_13 U6_X #2移载Y轴压装位
LD TR0
AND 1010.03  ; RK_13 U6_X #2移载Y轴#1轮廓检测位设定确认
MOVL(498) E1_356 E1_2226  ; RK_13 U6_X #2移载Y轴轴当前位置, RK_13 U6_X #2移载Y轴#1轮廓检测位
LD TR0
AND 1010.04  ; RK_13 U6_X #2移载Y轴#2轮廓检测位设定确认
MOVL(498) E1_356 E1_2228  ; RK_13 U6_X #2移载Y轴轴当前位置, RK_13 U6_X #2移载Y轴#2轮廓检测位
LD TR0
AND 1010.05  ; RK_13 U6_X #2移载Y轴激光焊接位设定确认
MOVL(498) E1_356 E1_2230  ; RK_13 U6_X #2移载Y轴轴当前位置, RK_13 U6_X #2移载Y轴激光焊接位
; rung 8: RK_13 U6_X #2移载Y轴运行条件
LDNOT 812.08  ; RK_13 U6_X #2移载Y轴报警信号标志[0012.08]
AND 812.09  ; RK_13 U6_X #2移载Y轴准备好了信号标志[0012.09]
ANDNOT 200.01  ; 紧急停止
ANDNOT 2060.15  ; RK_13 U6_X #2移载Y轴停止
OUT D1252.00  ; RK_13 U6_X #2移载Y轴运行条件

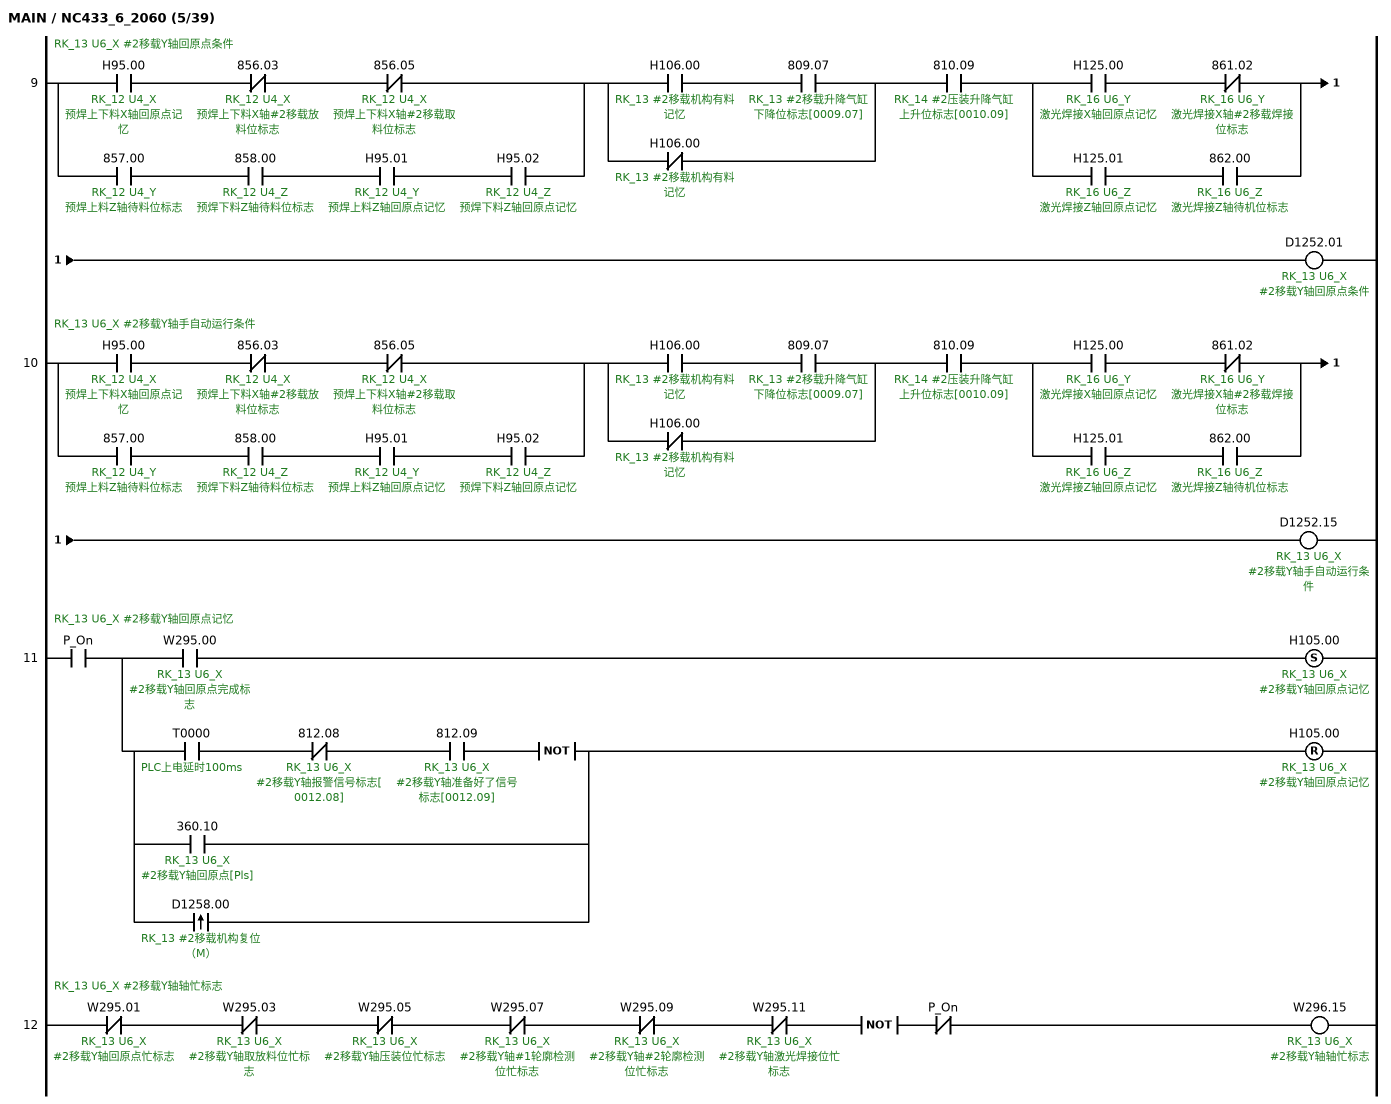
; rung 9: RK_13 U6_X #2移载Y轴回原点条件
LD H95.00  ; RK_12 U4_X 预焊上下料X轴回原点记忆
ANDNOT 856.03  ; RK_12 U4_X 预焊上下料X轴#2移载放料位标志
ANDNOT 856.05  ; RK_12 U4_X 预焊上下料X轴#2移载取料位标志
LD 857.00  ; RK_12 U4_Y 预焊上料Z轴待料位标志
AND 858.00  ; RK_12 U4_Z 预焊下料Z轴待料位标志
AND H95.01  ; RK_12 U4_Y 预焊上料Z轴回原点记忆
AND H95.02  ; RK_12 U4_Z 预焊下料Z轴回原点记忆
ORLD
LD H106.00  ; RK_13 #2移载机构有料记忆
AND 809.07  ; RK_13 #2移载升降气缸下降位标志[0009.07]
ORNOT H106.00  ; RK_13 #2移载机构有料记忆
ANDLD
AND 810.09  ; RK_14 #2压装升降气缸上升位标志[0010.09]
LD H125.00  ; RK_16 U6_Y 激光焊接X轴回原点记忆
ANDNOT 861.02  ; RK_16 U6_Y 激光焊接X轴#2移载焊接位标志
LD H125.01  ; RK_16 U6_Z 激光焊接Z轴回原点记忆
AND 862.00  ; RK_16 U6_Z 激光焊接Z轴待机位标志
ORLD
ANDLD
OUT D1252.01  ; RK_13 U6_X #2移载Y轴回原点条件
; rung 10: RK_13 U6_X #2移载Y轴手自动运行条件
LD H95.00  ; RK_12 U4_X 预焊上下料X轴回原点记忆
ANDNOT 856.03  ; RK_12 U4_X 预焊上下料X轴#2移载放料位标志
ANDNOT 856.05  ; RK_12 U4_X 预焊上下料X轴#2移载取料位标志
LD 857.00  ; RK_12 U4_Y 预焊上料Z轴待料位标志
AND 858.00  ; RK_12 U4_Z 预焊下料Z轴待料位标志
AND H95.01  ; RK_12 U4_Y 预焊上料Z轴回原点记忆
AND H95.02  ; RK_12 U4_Z 预焊下料Z轴回原点记忆
ORLD
LD H106.00  ; RK_13 #2移载机构有料记忆
AND 809.07  ; RK_13 #2移载升降气缸下降位标志[0009.07]
ORNOT H106.00  ; RK_13 #2移载机构有料记忆
ANDLD
AND 810.09  ; RK_14 #2压装升降气缸上升位标志[0010.09]
LD H125.00  ; RK_16 U6_Y 激光焊接X轴回原点记忆
ANDNOT 861.02  ; RK_16 U6_Y 激光焊接X轴#2移载焊接位标志
LD H125.01  ; RK_16 U6_Z 激光焊接Z轴回原点记忆
AND 862.00  ; RK_16 U6_Z 激光焊接Z轴待机位标志
ORLD
ANDLD
OUT D1252.15  ; RK_13 U6_X #2移载Y轴手自动运行条件
; rung 11: RK_13 U6_X #2移载Y轴回原点记忆
LD P_On
OUT TR0
AND W295.00  ; RK_13 U6_X #2移载Y轴回原点完成标志
SET H105.00  ; RK_13 U6_X #2移载Y轴回原点记忆
LD TR0
LD T0000  ; PLC上电延时100ms
ANDNOT 812.08  ; RK_13 U6_X #2移载Y轴报警信号标志[0012.08]
AND 812.09  ; RK_13 U6_X #2移载Y轴准备好了信号标志[0012.09]
NOT(520)
OR 360.10  ; RK_13 U6_X #2移载Y轴回原点[Pls]
@OR D1258.00  ; RK_13 #2移载机构复位（M）
ANDLD
RSET H105.00  ; RK_13 U6_X #2移载Y轴回原点记忆
; rung 12: RK_13 U6_X #2移载Y轴轴忙标志
LDNOT W295.01  ; RK_13 U6_X #2移载Y轴回原点忙标志
ANDNOT W295.03  ; RK_13 U6_X #2移载Y轴取放料位忙标志
ANDNOT W295.05  ; RK_13 U6_X #2移载Y轴压装位忙标志
ANDNOT W295.07  ; RK_13 U6_X #2移载Y轴#1轮廓检测位忙标志
ANDNOT W295.09  ; RK_13 U6_X #2移载Y轴#2轮廓检测位忙标志
ANDNOT W295.11  ; RK_13 U6_X #2移载Y轴激光焊接位忙标志
NOT(520)
ANDNOT P_On
OUT W296.15  ; RK_13 U6_X #2移载Y轴轴忙标志

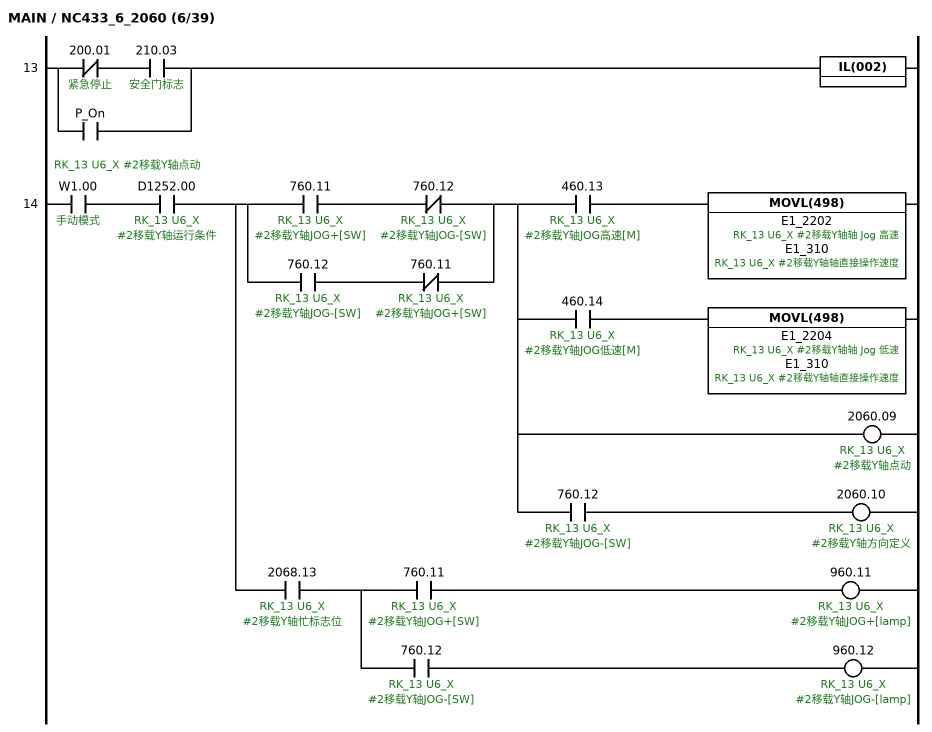
; rung 13
LDNOT 200.01  ; 紧急停止
AND 210.03  ; 安全门标志
OR P_On
IL(002)
; rung 14: RK_13 U6_X #2移载Y轴点动
LD W1.00  ; 手动模式
AND D1252.00  ; RK_13 U6_X #2移载Y轴运行条件
OUT TR0
LD 760.11  ; RK_13 U6_X #2移载Y轴JOG+[SW]
ANDNOT 760.12  ; RK_13 U6_X #2移载Y轴JOG-[SW]
LD 760.12  ; RK_13 U6_X #2移载Y轴JOG-[SW]
ANDNOT 760.11  ; RK_13 U6_X #2移载Y轴JOG+[SW]
ORLD
ANDLD
OUT TR1
AND 460.13  ; RK_13 U6_X #2移载Y轴JOG高速[M]
MOVL(498) E1_2202 E1_310  ; RK_13 U6_X #2移载Y轴轴 Jog 高速, RK_13 U6_X #2移载Y轴轴直接操作速度
LD TR1
AND 460.14  ; RK_13 U6_X #2移载Y轴JOG低速[M]
MOVL(498) E1_2204 E1_310  ; RK_13 U6_X #2移载Y轴轴 Jog 低速, RK_13 U6_X #2移载Y轴轴直接操作速度
LD TR1
OUT 2060.09  ; RK_13 U6_X #2移载Y轴点动
AND 760.12  ; RK_13 U6_X #2移载Y轴JOG-[SW]
OUT 2060.10  ; RK_13 U6_X #2移载Y轴方向定义
LD TR0
AND 2068.13  ; RK_13 U6_X #2移载Y轴忙标志位
OUT TR0
AND 760.11  ; RK_13 U6_X #2移载Y轴JOG+[SW]
OUT 960.11  ; RK_13 U6_X #2移载Y轴JOG+[lamp]
LD TR0
AND 760.12  ; RK_13 U6_X #2移载Y轴JOG-[SW]
OUT 960.12  ; RK_13 U6_X #2移载Y轴JOG-[lamp]

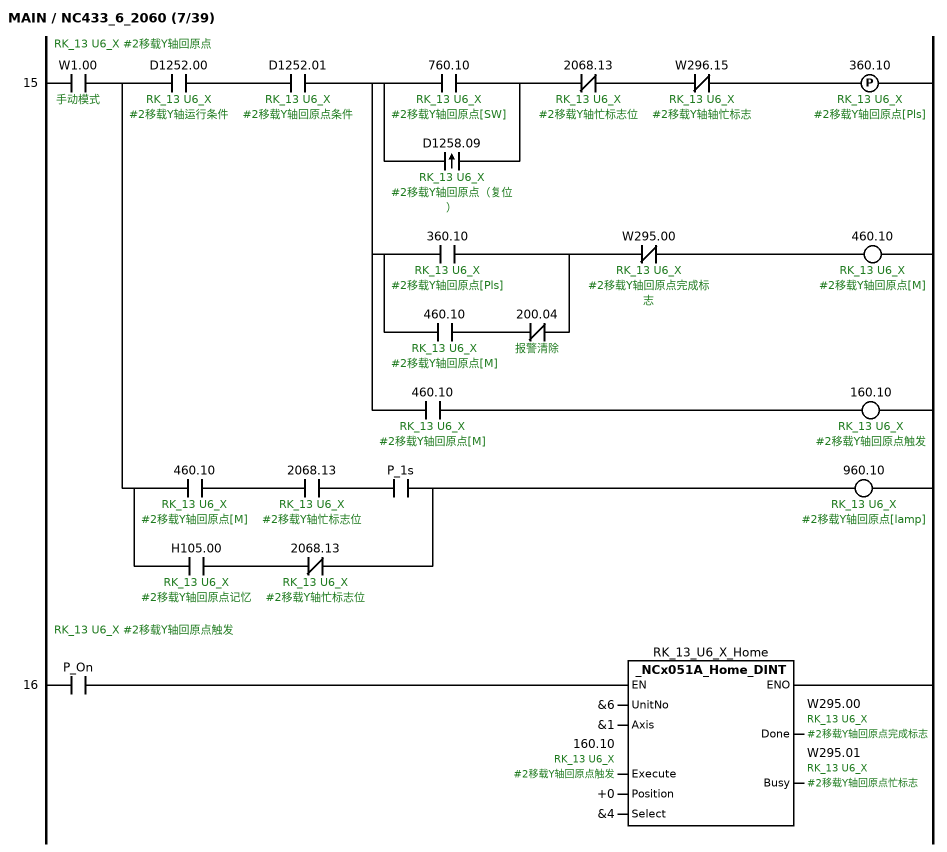
; rung 15: RK_13 U6_X #2移载Y轴回原点
LD W1.00  ; 手动模式
OUT TR0
AND D1252.00  ; RK_13 U6_X #2移载Y轴运行条件
AND D1252.01  ; RK_13 U6_X #2移载Y轴回原点条件
OUT TR1
LD 760.10  ; RK_13 U6_X #2移载Y轴回原点[SW]
@OR D1258.09  ; RK_13 U6_X #2移载Y轴回原点（复位）
ANDLD
ANDNOT 2068.13  ; RK_13 U6_X #2移载Y轴忙标志位
ANDNOT W296.15  ; RK_13 U6_X #2移载Y轴轴忙标志
DIFU(013) 360.10  ; RK_13 U6_X #2移载Y轴回原点[Pls]
LD TR1
LD 360.10  ; RK_13 U6_X #2移载Y轴回原点[Pls]
LD 460.10  ; RK_13 U6_X #2移载Y轴回原点[M]
ANDNOT 200.04  ; 报警清除
ORLD
ANDLD
ANDNOT W295.00  ; RK_13 U6_X #2移载Y轴回原点完成标志
OUT 460.10  ; RK_13 U6_X #2移载Y轴回原点[M]
LD TR1
AND 460.10  ; RK_13 U6_X #2移载Y轴回原点[M]
OUT 160.10  ; RK_13 U6_X #2移载Y轴回原点触发
LD TR0
LD 460.10  ; RK_13 U6_X #2移载Y轴回原点[M]
AND 2068.13  ; RK_13 U6_X #2移载Y轴忙标志位
AND P_1s
LD H105.00  ; RK_13 U6_X #2移载Y轴回原点记忆
ANDNOT 2068.13  ; RK_13 U6_X #2移载Y轴忙标志位
ORLD
ANDLD
OUT 960.10  ; RK_13 U6_X #2移载Y轴回原点[lamp]
; rung 16: RK_13 U6_X #2移载Y轴回原点触发
LD P_On
CALL RK_13_U6_X_Home : _NCx051A_Home_DINT (UnitNo := &6, Axis := &1, Execute := 160.10, Position := +0, Select := &4, Done => W295.00, Busy => W295.01)  ; RK_13 U6_X #2移载Y轴回原点触发, RK_13 U6_X #2移载Y轴回原点完成标志, RK_13 U6_X #2移载Y轴回原点忙标志

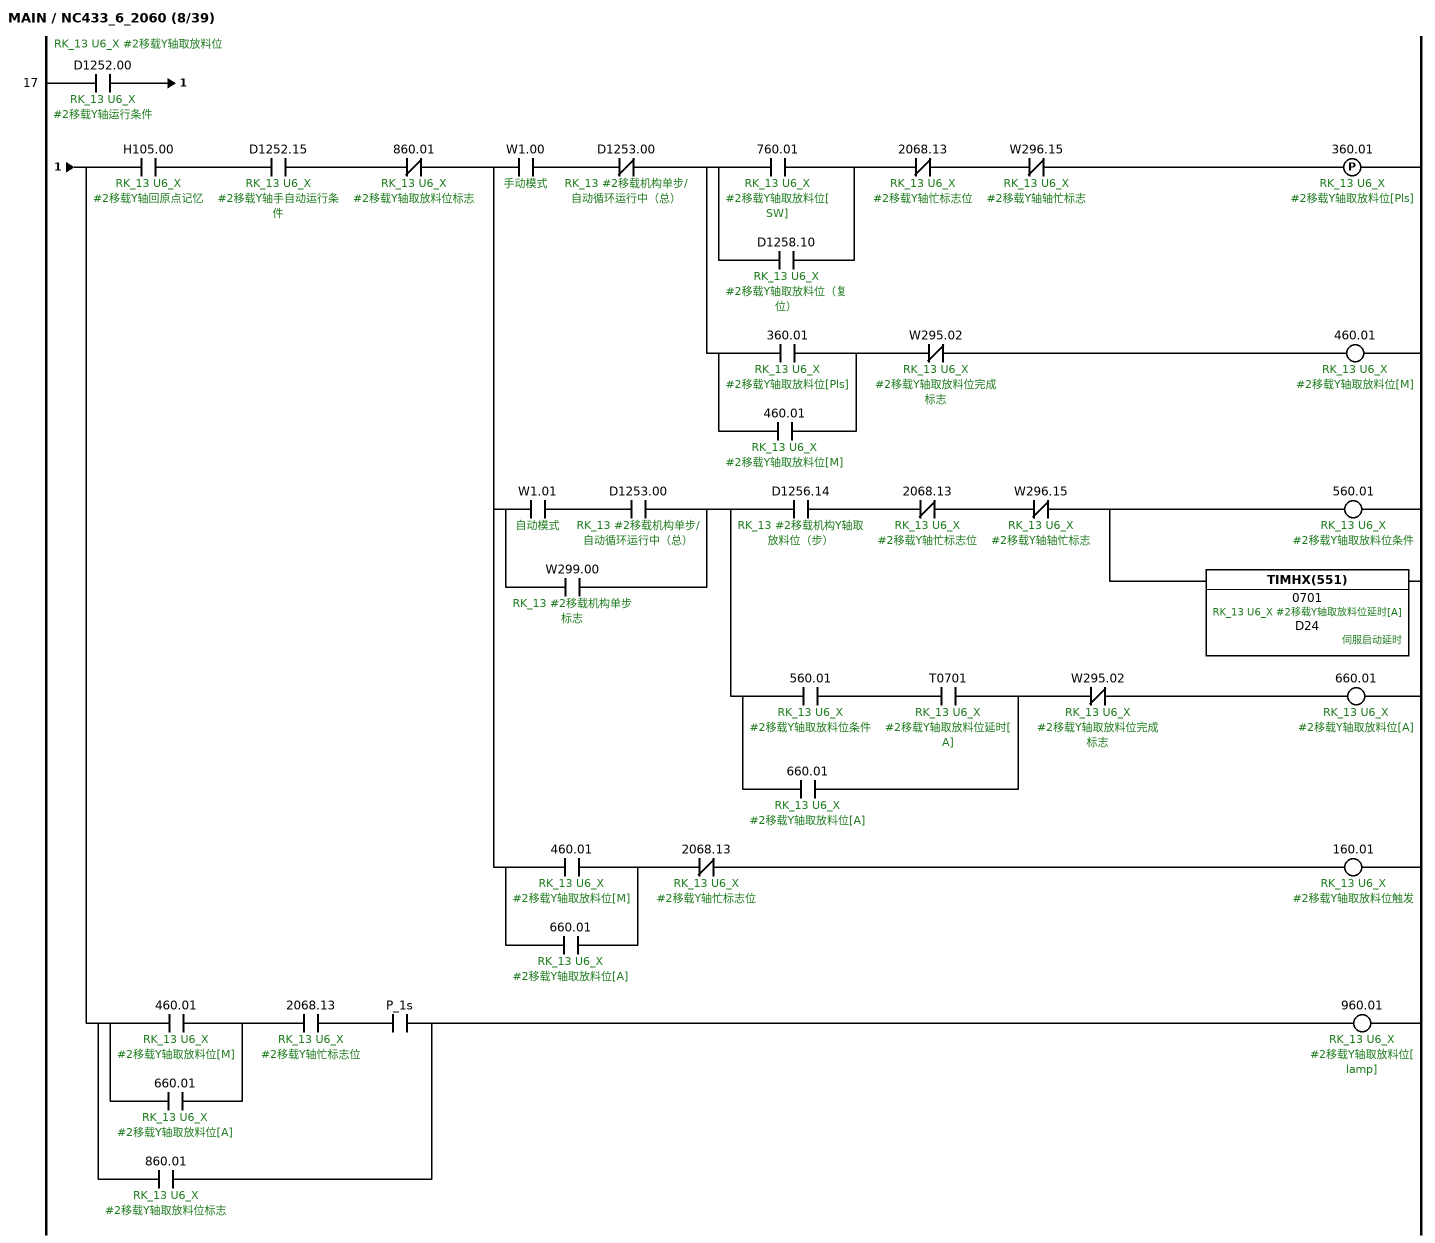
; rung 17: RK_13 U6_X #2移载Y轴取放料位
LD D1252.00  ; RK_13 U6_X #2移载Y轴运行条件
OUT TR0
AND H105.00  ; RK_13 U6_X #2移载Y轴回原点记忆
AND D1252.15  ; RK_13 U6_X #2移载Y轴手自动运行条件
ANDNOT 860.01  ; RK_13 U6_X #2移载Y轴取放料位标志
OUT TR1
AND W1.00  ; 手动模式
ANDNOT D1253.00  ; RK_13 #2移载机构单步/自动循环运行中（总）
OUT TR2
LD 760.01  ; RK_13 U6_X #2移载Y轴取放料位[SW]
OR D1258.10  ; RK_13 U6_X #2移载Y轴取放料位（复位）
ANDLD
ANDNOT 2068.13  ; RK_13 U6_X #2移载Y轴忙标志位
ANDNOT W296.15  ; RK_13 U6_X #2移载Y轴轴忙标志
DIFU(013) 360.01  ; RK_13 U6_X #2移载Y轴取放料位[Pls]
LD TR2
LD 360.01  ; RK_13 U6_X #2移载Y轴取放料位[Pls]
OR 460.01  ; RK_13 U6_X #2移载Y轴取放料位[M]
ANDLD
ANDNOT W295.02  ; RK_13 U6_X #2移载Y轴取放料位完成标志
OUT 460.01  ; RK_13 U6_X #2移载Y轴取放料位[M]
LD TR1
LD W1.01  ; 自动模式
AND D1253.00  ; RK_13 #2移载机构单步/自动循环运行中（总）
OR W299.00  ; RK_13 #2移载机构单步标志
ANDLD
OUT TR2
AND D1256.14  ; RK_13 #2移载机构Y轴取放料位（步）
ANDNOT 2068.13  ; RK_13 U6_X #2移载Y轴忙标志位
ANDNOT W296.15  ; RK_13 U6_X #2移载Y轴轴忙标志
OUT 560.01  ; RK_13 U6_X #2移载Y轴取放料位条件
TIMHX(551) 0701 D24  ; 伺服启动延时, RK_13 U6_X #2移载Y轴取放料位延时[A]
LD TR2
LD 560.01  ; RK_13 U6_X #2移载Y轴取放料位条件
AND T0701  ; RK_13 U6_X #2移载Y轴取放料位延时[A]
OR 660.01  ; RK_13 U6_X #2移载Y轴取放料位[A]
ANDLD
ANDNOT W295.02  ; RK_13 U6_X #2移载Y轴取放料位完成标志
OUT 660.01  ; RK_13 U6_X #2移载Y轴取放料位[A]
LD TR1
LD 460.01  ; RK_13 U6_X #2移载Y轴取放料位[M]
OR 660.01  ; RK_13 U6_X #2移载Y轴取放料位[A]
ANDLD
ANDNOT 2068.13  ; RK_13 U6_X #2移载Y轴忙标志位
OUT 160.01  ; RK_13 U6_X #2移载Y轴取放料位触发
LD TR0
LD 460.01  ; RK_13 U6_X #2移载Y轴取放料位[M]
OR 660.01  ; RK_13 U6_X #2移载Y轴取放料位[A]
AND 2068.13  ; RK_13 U6_X #2移载Y轴忙标志位
AND P_1s
OR 860.01  ; RK_13 U6_X #2移载Y轴取放料位标志
ANDLD
OUT 960.01  ; RK_13 U6_X #2移载Y轴取放料位[lamp]

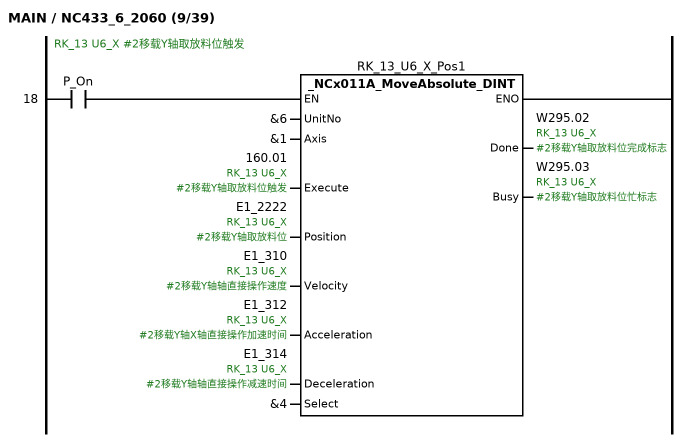
; rung 18: RK_13 U6_X #2移载Y轴取放料位触发
LD P_On
CALL RK_13_U6_X_Pos1 : _NCx011A_MoveAbsolute_DINT (UnitNo := &6, Axis := &1, Execute := 160.01, Position := E1_2222, Velocity := E1_310, Acceleration := E1_312, Deceleration := E1_314, Select := &4, Done => W295.02, Busy => W295.03)  ; RK_13 U6_X #2移载Y轴取放料位触发, RK_13 U6_X #2移载Y轴取放料位, RK_13 U6_X #2移载Y轴轴直接操作速度, RK_13 U6_X #2移载Y轴X轴直接操作加速时间, RK_13 U6_X #2移载Y轴轴直接操作减速时间, RK_13 U6_X #2移载Y轴取放料位完成标志, RK_13 U6_X #2移载Y轴取放料位忙标志

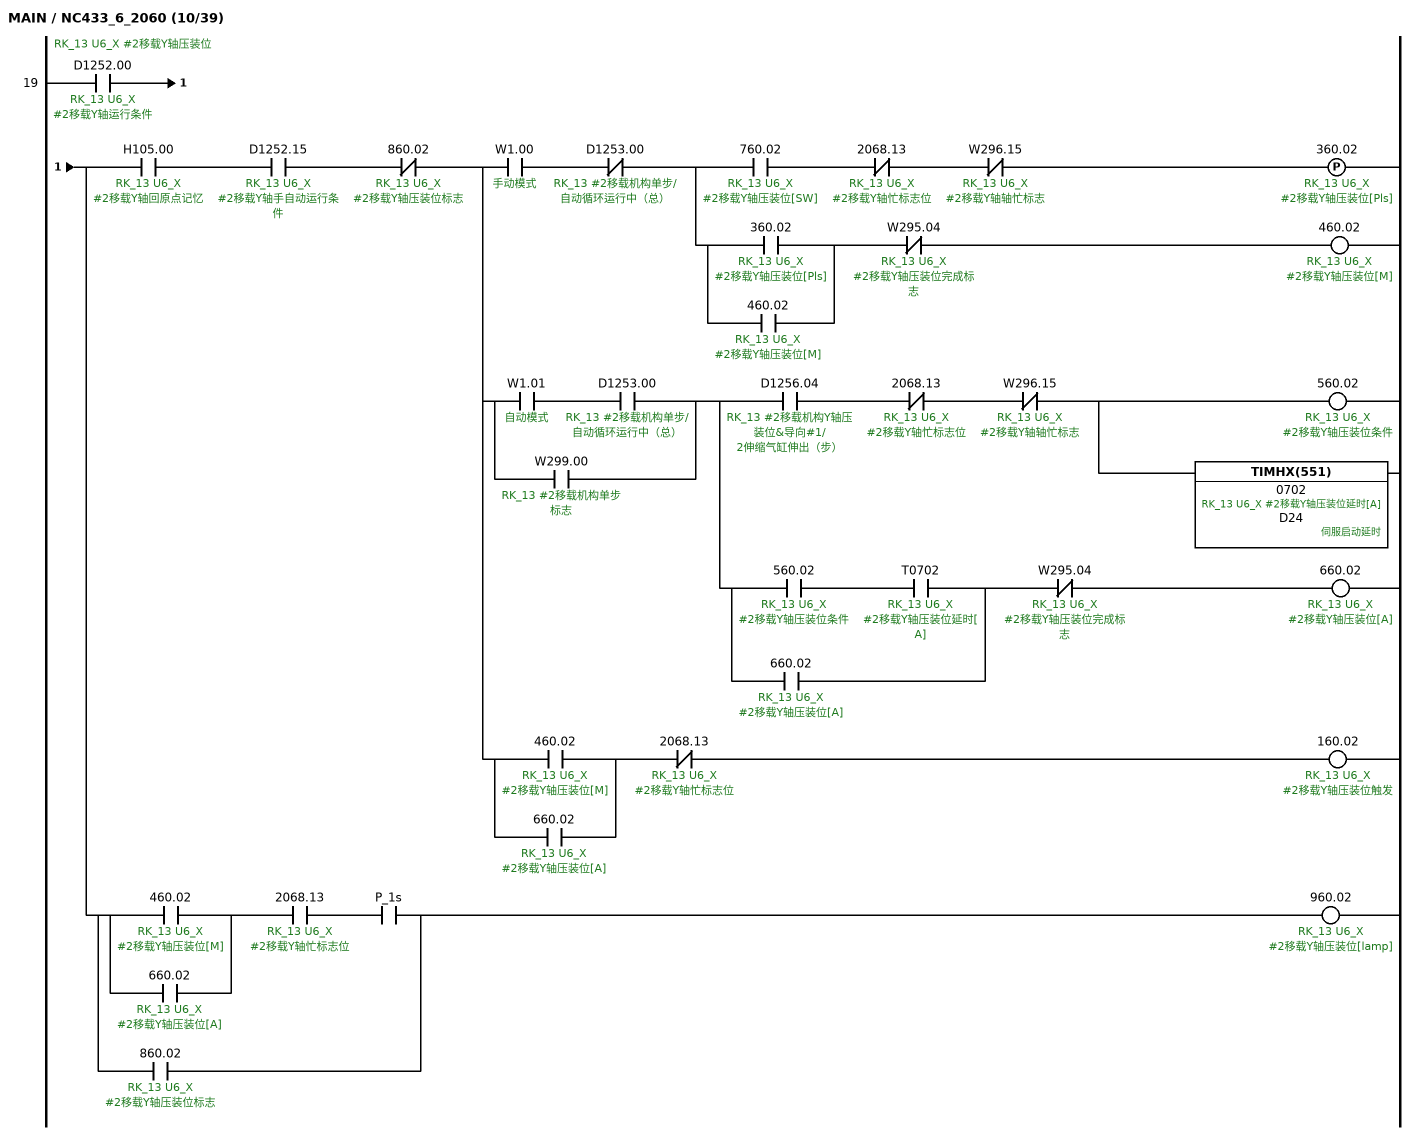
; rung 19: RK_13 U6_X #2移载Y轴压装位
LD D1252.00  ; RK_13 U6_X #2移载Y轴运行条件
OUT TR0
AND H105.00  ; RK_13 U6_X #2移载Y轴回原点记忆
AND D1252.15  ; RK_13 U6_X #2移载Y轴手自动运行条件
ANDNOT 860.02  ; RK_13 U6_X #2移载Y轴压装位标志
OUT TR1
AND W1.00  ; 手动模式
ANDNOT D1253.00  ; RK_13 #2移载机构单步/自动循环运行中（总）
OUT TR2
AND 760.02  ; RK_13 U6_X #2移载Y轴压装位[SW]
ANDNOT 2068.13  ; RK_13 U6_X #2移载Y轴忙标志位
ANDNOT W296.15  ; RK_13 U6_X #2移载Y轴轴忙标志
DIFU(013) 360.02  ; RK_13 U6_X #2移载Y轴压装位[Pls]
LD TR2
LD 360.02  ; RK_13 U6_X #2移载Y轴压装位[Pls]
OR 460.02  ; RK_13 U6_X #2移载Y轴压装位[M]
ANDLD
ANDNOT W295.04  ; RK_13 U6_X #2移载Y轴压装位完成标志
OUT 460.02  ; RK_13 U6_X #2移载Y轴压装位[M]
LD TR1
LD W1.01  ; 自动模式
AND D1253.00  ; RK_13 #2移载机构单步/自动循环运行中（总）
OR W299.00  ; RK_13 #2移载机构单步标志
ANDLD
OUT TR2
AND D1256.04  ; RK_13 #2移载机构Y轴压装位&导向#1/2伸缩气缸伸出（步）
ANDNOT 2068.13  ; RK_13 U6_X #2移载Y轴忙标志位
ANDNOT W296.15  ; RK_13 U6_X #2移载Y轴轴忙标志
OUT 560.02  ; RK_13 U6_X #2移载Y轴压装位条件
TIMHX(551) 0702 D24  ; 伺服启动延时, RK_13 U6_X #2移载Y轴压装位延时[A]
LD TR2
LD 560.02  ; RK_13 U6_X #2移载Y轴压装位条件
AND T0702  ; RK_13 U6_X #2移载Y轴压装位延时[A]
OR 660.02  ; RK_13 U6_X #2移载Y轴压装位[A]
ANDLD
ANDNOT W295.04  ; RK_13 U6_X #2移载Y轴压装位完成标志
OUT 660.02  ; RK_13 U6_X #2移载Y轴压装位[A]
LD TR1
LD 460.02  ; RK_13 U6_X #2移载Y轴压装位[M]
OR 660.02  ; RK_13 U6_X #2移载Y轴压装位[A]
ANDLD
ANDNOT 2068.13  ; RK_13 U6_X #2移载Y轴忙标志位
OUT 160.02  ; RK_13 U6_X #2移载Y轴压装位触发
LD TR0
LD 460.02  ; RK_13 U6_X #2移载Y轴压装位[M]
OR 660.02  ; RK_13 U6_X #2移载Y轴压装位[A]
AND 2068.13  ; RK_13 U6_X #2移载Y轴忙标志位
AND P_1s
OR 860.02  ; RK_13 U6_X #2移载Y轴压装位标志
ANDLD
OUT 960.02  ; RK_13 U6_X #2移载Y轴压装位[lamp]

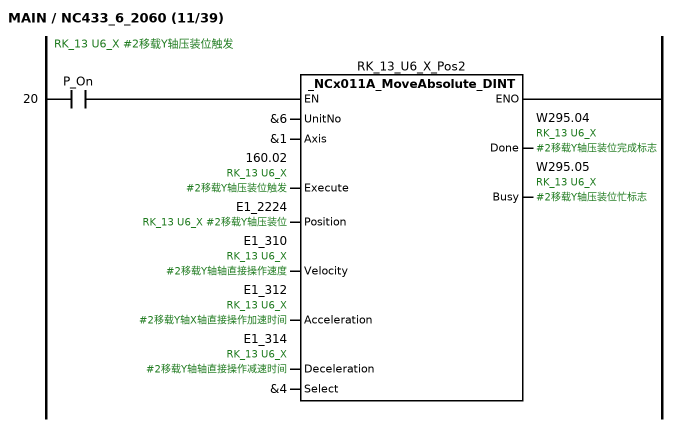
; rung 20: RK_13 U6_X #2移载Y轴压装位触发
LD P_On
CALL RK_13_U6_X_Pos2 : _NCx011A_MoveAbsolute_DINT (UnitNo := &6, Axis := &1, Execute := 160.02, Position := E1_2224, Velocity := E1_310, Acceleration := E1_312, Deceleration := E1_314, Select := &4, Done => W295.04, Busy => W295.05)  ; RK_13 U6_X #2移载Y轴压装位触发, RK_13 U6_X #2移载Y轴压装位, RK_13 U6_X #2移载Y轴轴直接操作速度, RK_13 U6_X #2移载Y轴X轴直接操作加速时间, RK_13 U6_X #2移载Y轴轴直接操作减速时间, RK_13 U6_X #2移载Y轴压装位完成标志, RK_13 U6_X #2移载Y轴压装位忙标志

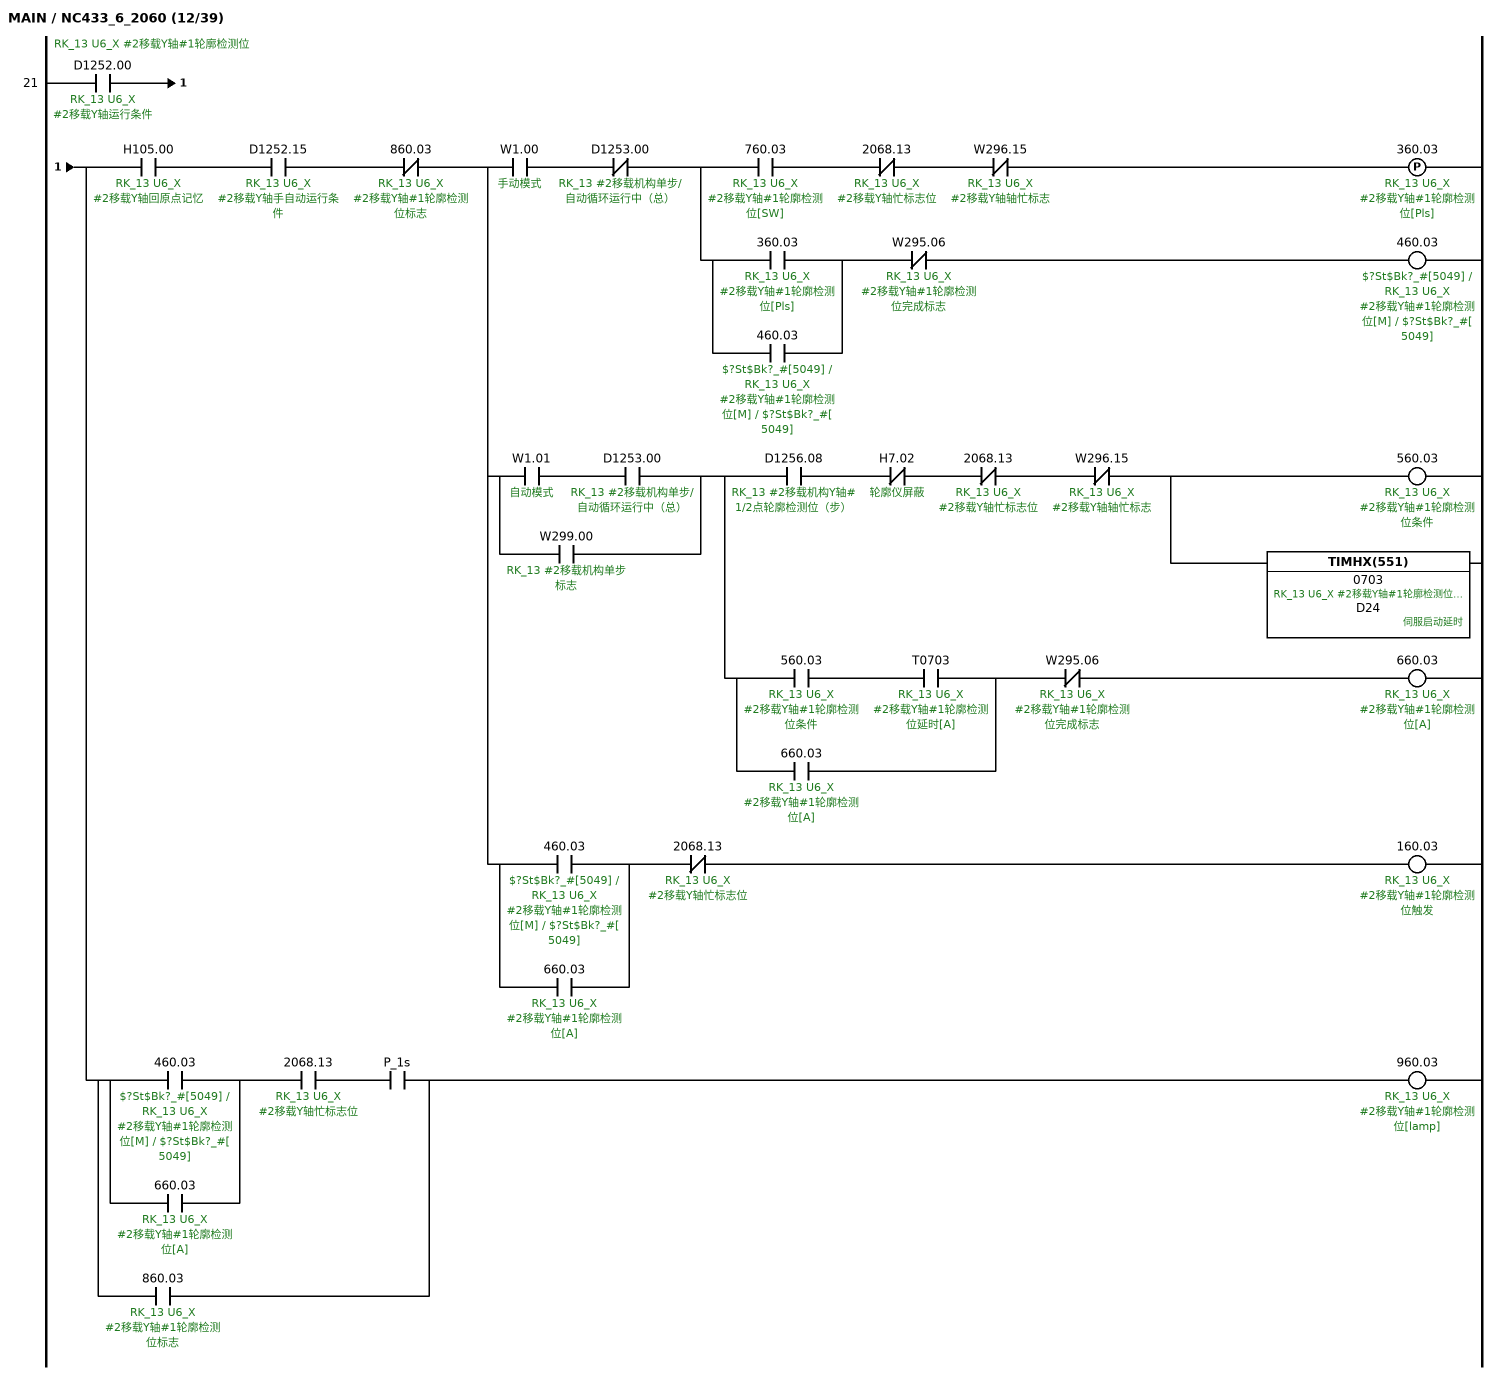
; rung 21: RK_13 U6_X #2移载Y轴#1轮廓检测位
LD D1252.00  ; RK_13 U6_X #2移载Y轴运行条件
OUT TR0
AND H105.00  ; RK_13 U6_X #2移载Y轴回原点记忆
AND D1252.15  ; RK_13 U6_X #2移载Y轴手自动运行条件
ANDNOT 860.03  ; RK_13 U6_X #2移载Y轴#1轮廓检测位标志
OUT TR1
AND W1.00  ; 手动模式
ANDNOT D1253.00  ; RK_13 #2移载机构单步/自动循环运行中（总）
OUT TR2
AND 760.03  ; RK_13 U6_X #2移载Y轴#1轮廓检测位[SW]
ANDNOT 2068.13  ; RK_13 U6_X #2移载Y轴忙标志位
ANDNOT W296.15  ; RK_13 U6_X #2移载Y轴轴忙标志
DIFU(013) 360.03  ; RK_13 U6_X #2移载Y轴#1轮廓检测位[Pls]
LD TR2
LD 360.03  ; RK_13 U6_X #2移载Y轴#1轮廓检测位[Pls]
OR 460.03  ; $?St$Bk?_#[5049] / RK_13 U6_X #2移载Y轴#1轮廓检测位[M] / $?St$Bk?_#[5049]
ANDLD
ANDNOT W295.06  ; RK_13 U6_X #2移载Y轴#1轮廓检测位完成标志
OUT 460.03  ; $?St$Bk?_#[5049] / RK_13 U6_X #2移载Y轴#1轮廓检测位[M] / $?St$Bk?_#[5049]
LD TR1
LD W1.01  ; 自动模式
AND D1253.00  ; RK_13 #2移载机构单步/自动循环运行中（总）
OR W299.00  ; RK_13 #2移载机构单步标志
ANDLD
OUT TR2
AND D1256.08  ; RK_13 #2移载机构Y轴#1/2点轮廓检测位（步）
ANDNOT H7.02  ; 轮廓仪屏蔽
ANDNOT 2068.13  ; RK_13 U6_X #2移载Y轴忙标志位
ANDNOT W296.15  ; RK_13 U6_X #2移载Y轴轴忙标志
OUT 560.03  ; RK_13 U6_X #2移载Y轴#1轮廓检测位条件
TIMHX(551) 0703 D24  ; 伺服启动延时, RK_13 U6_X #2移载Y轴#1轮廓检测位延时[A]
LD TR2
LD 560.03  ; RK_13 U6_X #2移载Y轴#1轮廓检测位条件
AND T0703  ; RK_13 U6_X #2移载Y轴#1轮廓检测位延时[A]
OR 660.03  ; RK_13 U6_X #2移载Y轴#1轮廓检测位[A]
ANDLD
ANDNOT W295.06  ; RK_13 U6_X #2移载Y轴#1轮廓检测位完成标志
OUT 660.03  ; RK_13 U6_X #2移载Y轴#1轮廓检测位[A]
LD TR1
LD 460.03  ; $?St$Bk?_#[5049] / RK_13 U6_X #2移载Y轴#1轮廓检测位[M] / $?St$Bk?_#[5049]
OR 660.03  ; RK_13 U6_X #2移载Y轴#1轮廓检测位[A]
ANDLD
ANDNOT 2068.13  ; RK_13 U6_X #2移载Y轴忙标志位
OUT 160.03  ; RK_13 U6_X #2移载Y轴#1轮廓检测位触发
LD TR0
LD 460.03  ; $?St$Bk?_#[5049] / RK_13 U6_X #2移载Y轴#1轮廓检测位[M] / $?St$Bk?_#[5049]
OR 660.03  ; RK_13 U6_X #2移载Y轴#1轮廓检测位[A]
AND 2068.13  ; RK_13 U6_X #2移载Y轴忙标志位
AND P_1s
OR 860.03  ; RK_13 U6_X #2移载Y轴#1轮廓检测位标志
ANDLD
OUT 960.03  ; RK_13 U6_X #2移载Y轴#1轮廓检测位[lamp]

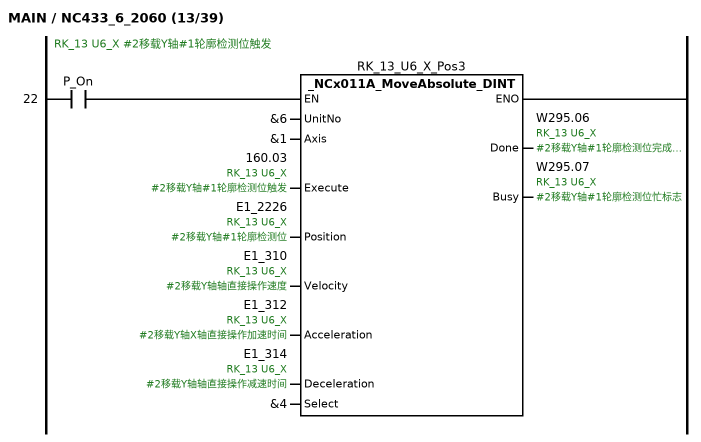
; rung 22: RK_13 U6_X #2移载Y轴#1轮廓检测位触发
LD P_On
CALL RK_13_U6_X_Pos3 : _NCx011A_MoveAbsolute_DINT (UnitNo := &6, Axis := &1, Execute := 160.03, Position := E1_2226, Velocity := E1_310, Acceleration := E1_312, Deceleration := E1_314, Select := &4, Done => W295.06, Busy => W295.07)  ; RK_13 U6_X #2移载Y轴#1轮廓检测位触发, RK_13 U6_X #2移载Y轴#1轮廓检测位, RK_13 U6_X #2移载Y轴轴直接操作速度, RK_13 U6_X #2移载Y轴X轴直接操作加速时间, RK_13 U6_X #2移载Y轴轴直接操作减速时间, RK_13 U6_X #2移载Y轴#1轮廓检测位完成标志, RK_13 U6_X #2移载Y轴#1轮廓检测位忙标志

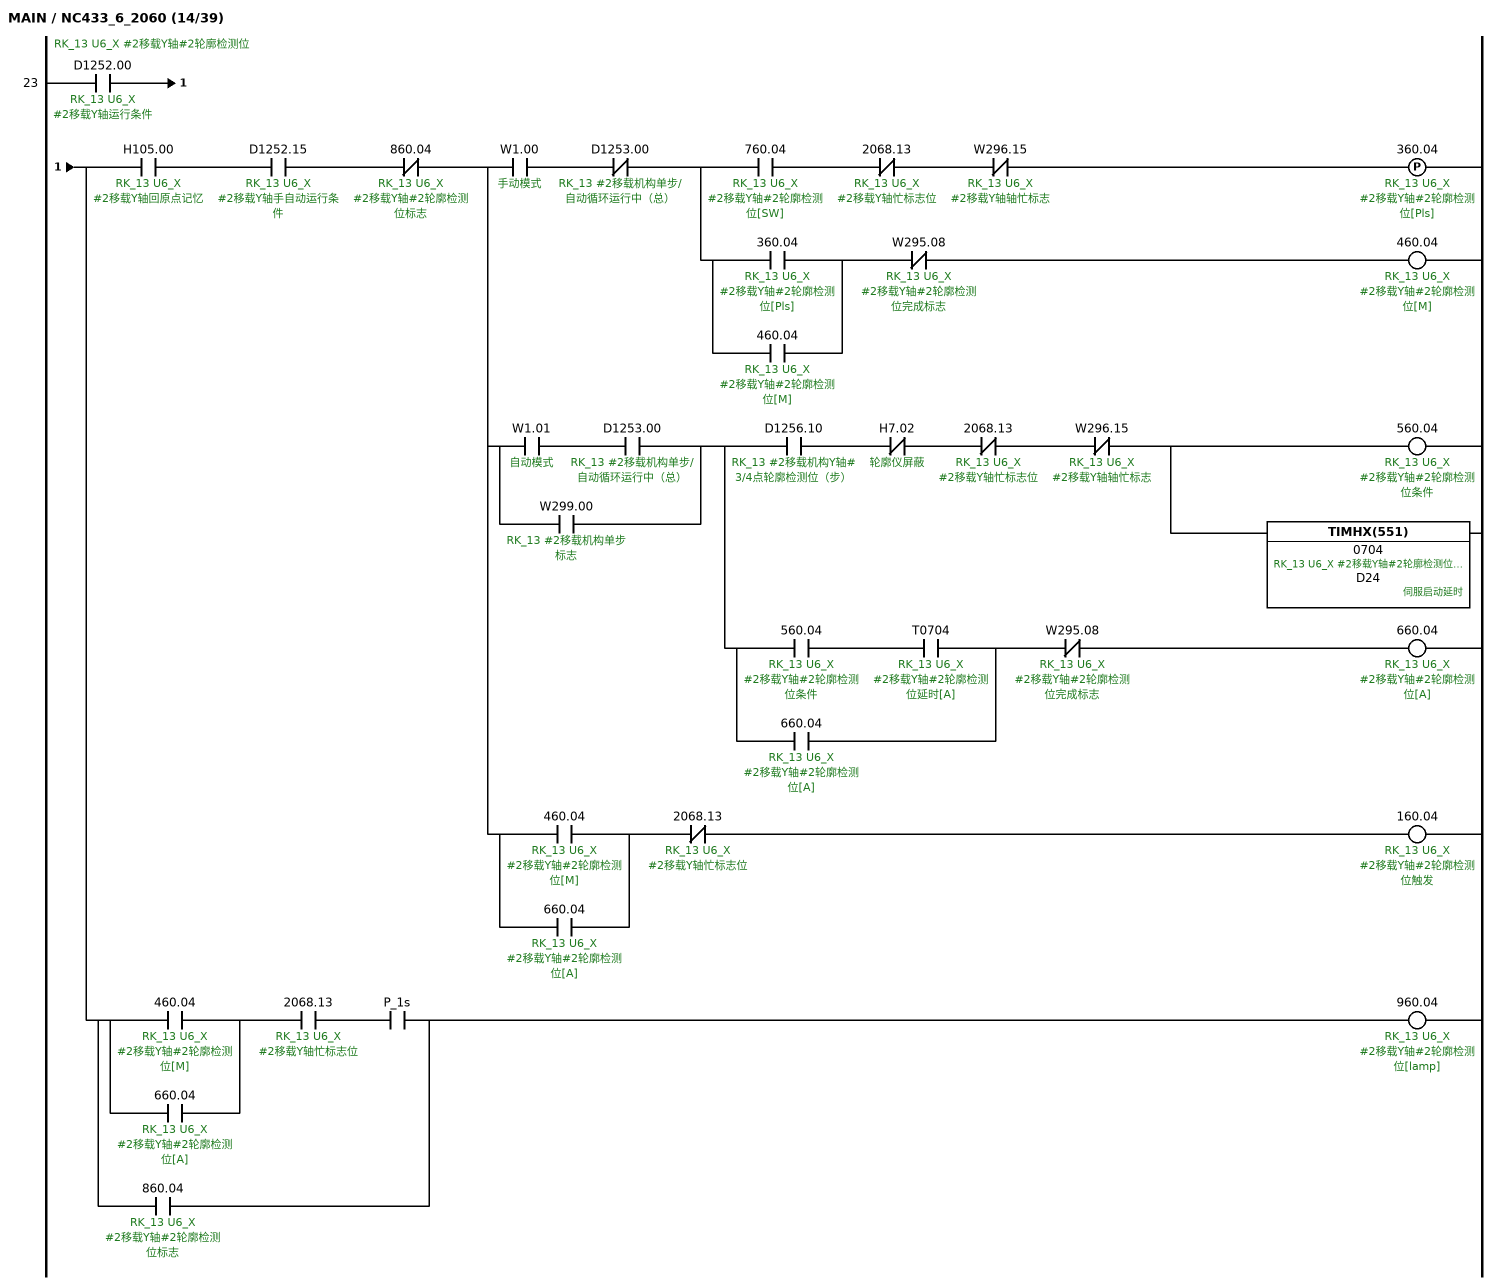
; rung 23: RK_13 U6_X #2移载Y轴#2轮廓检测位
LD D1252.00  ; RK_13 U6_X #2移载Y轴运行条件
OUT TR0
AND H105.00  ; RK_13 U6_X #2移载Y轴回原点记忆
AND D1252.15  ; RK_13 U6_X #2移载Y轴手自动运行条件
ANDNOT 860.04  ; RK_13 U6_X #2移载Y轴#2轮廓检测位标志
OUT TR1
AND W1.00  ; 手动模式
ANDNOT D1253.00  ; RK_13 #2移载机构单步/自动循环运行中（总）
OUT TR2
AND 760.04  ; RK_13 U6_X #2移载Y轴#2轮廓检测位[SW]
ANDNOT 2068.13  ; RK_13 U6_X #2移载Y轴忙标志位
ANDNOT W296.15  ; RK_13 U6_X #2移载Y轴轴忙标志
DIFU(013) 360.04  ; RK_13 U6_X #2移载Y轴#2轮廓检测位[Pls]
LD TR2
LD 360.04  ; RK_13 U6_X #2移载Y轴#2轮廓检测位[Pls]
OR 460.04  ; RK_13 U6_X #2移载Y轴#2轮廓检测位[M]
ANDLD
ANDNOT W295.08  ; RK_13 U6_X #2移载Y轴#2轮廓检测位完成标志
OUT 460.04  ; RK_13 U6_X #2移载Y轴#2轮廓检测位[M]
LD TR1
LD W1.01  ; 自动模式
AND D1253.00  ; RK_13 #2移载机构单步/自动循环运行中（总）
OR W299.00  ; RK_13 #2移载机构单步标志
ANDLD
OUT TR2
AND D1256.10  ; RK_13 #2移载机构Y轴#3/4点轮廓检测位（步）
ANDNOT H7.02  ; 轮廓仪屏蔽
ANDNOT 2068.13  ; RK_13 U6_X #2移载Y轴忙标志位
ANDNOT W296.15  ; RK_13 U6_X #2移载Y轴轴忙标志
OUT 560.04  ; RK_13 U6_X #2移载Y轴#2轮廓检测位条件
TIMHX(551) 0704 D24  ; 伺服启动延时, RK_13 U6_X #2移载Y轴#2轮廓检测位延时[A]
LD TR2
LD 560.04  ; RK_13 U6_X #2移载Y轴#2轮廓检测位条件
AND T0704  ; RK_13 U6_X #2移载Y轴#2轮廓检测位延时[A]
OR 660.04  ; RK_13 U6_X #2移载Y轴#2轮廓检测位[A]
ANDLD
ANDNOT W295.08  ; RK_13 U6_X #2移载Y轴#2轮廓检测位完成标志
OUT 660.04  ; RK_13 U6_X #2移载Y轴#2轮廓检测位[A]
LD TR1
LD 460.04  ; RK_13 U6_X #2移载Y轴#2轮廓检测位[M]
OR 660.04  ; RK_13 U6_X #2移载Y轴#2轮廓检测位[A]
ANDLD
ANDNOT 2068.13  ; RK_13 U6_X #2移载Y轴忙标志位
OUT 160.04  ; RK_13 U6_X #2移载Y轴#2轮廓检测位触发
LD TR0
LD 460.04  ; RK_13 U6_X #2移载Y轴#2轮廓检测位[M]
OR 660.04  ; RK_13 U6_X #2移载Y轴#2轮廓检测位[A]
AND 2068.13  ; RK_13 U6_X #2移载Y轴忙标志位
AND P_1s
OR 860.04  ; RK_13 U6_X #2移载Y轴#2轮廓检测位标志
ANDLD
OUT 960.04  ; RK_13 U6_X #2移载Y轴#2轮廓检测位[lamp]

